LIN {X 0,Y 162.27,Z 688.109,A -85,B 0,C 180,E1 -25954.265,E2 -25954.265} C_VEL
LIN {X 0,Y 156.818,Z 700.099,A -85,B 0,C 180,E1 -25956.224,E2 -25956.224} C_VEL
LIN {X 0,Y 150.778,Z 711.775,A -85,B 0,C 180,E1 -25958.67,E2 -25958.67} C_VEL
LIN {X 0,Y 143.94,Z 723.54,A -85,B 0,C 180,E1 -25961.874,E2 -25961.874} C_VEL
LIN {X 0,Y 137.759,Z 733.192,A -85,B 0,C 180,E1 -25965.296,E2 -25965.296} C_VEL
LIN {X 0,Y 132.844,Z 740.567,A -85,B 0,C 180,E1 -25968.599,E2 -25968.599} C_VEL
LIN {X 0,Y 126.818,Z 749.022,A -85,B 0,C 180,E1 -25973.433,E2 -25973.433} C_VEL
LIN {X 0,Y 121.728,Z 756.009,A -85,B 0,C 180,E1 -25978.692,E2 -25978.692} C_VEL
LIN {X 0,Y 117.214,Z 762.465,A -85,B 0,C 180,E1 -25985.182,E2 -25985.182} C_VEL
LIN {X 0,Y 114.114,Z 767.443,A -85,B 0,C 180,E1 -25992.063,E2 -25992.063} C_VEL
LIN {X 0,Y 112.508,Z 771.077,A -85,B 0,C 180,E1 -25999.197,E2 -25999.197} C_VEL
LIN {X 0,Y 112.216,Z 772.187,A -85,B 0,C 180,E1 -26002.183,E2 -26002.183} C_VEL
LIN {X 0,Y 111.418,Z 773.145,A -85,B 0,C 180,E1 -26005.137,E2 -26005.137} C_VEL
LIN {X 0,Y 109.742,Z 773.826,A -85,B 0,C 180,E1 -26008.075,E2 -26008.075} C_VEL
LIN {X 0,Y 106.019,Z 774.46,A -85,B 0,C 180,E1 -26014.176,E2 -26014.176} C_VEL
LIN {X 0,Y 105.123,Z 774.478,A -85,B 0,C 180,E1 -26017.421,E2 -26017.421} C_VEL
LIN {X 0,Y 105.117,Z 774.446,A -85,B 0,C 180,E1 -26018.519,E2 -26018.519} C_VEL
LIN {X 0,Y 106.239,Z 773.913,A -85,B 0,C 180,E1 -26025.342,E2 -26025.342} C_VEL
LIN {X 0,Y 108.989,Z 772.261,A -85,B 0,C 180,E1 -26032.759,E2 -26032.759} C_VEL
LIN {X 0,Y 113.268,Z 769.502,A -85,B 0,C 180,E1 -26039.758,E2 -26039.758} C_VEL
LIN {X 0,Y 119.195,Z 765.541,A -85,B 0,C 180,E1 -26046.127,E2 -26046.127} C_VEL
LIN {X 0,Y 126.402,Z 760.299,A -85,B 0,C 180,E1 -26051.849,E2 -26051.849} C_VEL
LIN {X 0,Y 132.654,Z 755.491,A -85,B 0,C 180,E1 -26055.659,E2 -26055.659} C_VEL
LIN {X 0,Y 139.26,Z 749.833,A -85,B 0,C 180,E1 -26059.197,E2 -26059.197} C_VEL
LIN {X 0,Y 147.754,Z 742.03,A -85,B 0,C 180,E1 -26062.815,E2 -26062.815} C_VEL
LIN {X 0,Y 156.831,Z 732.723,A -85,B 0,C 180,E1 -26065.996,E2 -26065.996} C_VEL
LIN {X 0,Y 166.319,Z 721.594,A -85,B 0,C 180,E1 -26068.832,E2 -26068.832} C_VEL
LIN {X 0,Y 174.952,Z 709.953,A -85,B 0,C 180,E1 -26071.034,E2 -26071.034} C_VEL
LIN {X 0,Y 182.722,Z 697.753,A -85,B 0,C 180,E1 -26072.801,E2 -26072.801} C_VEL
LIN {X 0,Y 190.165,Z 683.997,A -85,B 0,C 180,E1 -26074.264,E2 -26074.264} C_VEL
LIN {X 0,Y 196.216,Z 670.493,A -85,B 0,C 180,E1 -26075.346,E2 -26075.346} C_VEL
LIN {X 0,Y 201.613,Z 655.52,A -85,B 0,C 180,E1 -26076.208,E2 -26076.208} C_VEL
LIN {X 0,Y 205.675,Z 640.602,A -85,B 0,C 180,E1 -26076.834,E2 -26076.834} C_VEL
LIN {X 0,Y 208.57,Z 625.043,A -85,B 0,C 180,E1 -26077.319,E2 -26077.319} C_VEL
LIN {X 0,Y 212.506,Z 591.895,A -85,B 0,C 180,E1 -26078.08,E2 -26078.08} C_VEL
LIN {X 0,Y 212.507,Z 590.897,A -85,B 0,C 180,E1 -26078.239,E2 -26078.239} C_VEL
LIN {X 0,Y 211.324,Z 586.522,A -85,B 0,C 180,E1 -26080.576,E2 -26080.576} C_VEL
LIN {X 0,Y 210.411,Z 584.182,A -85,B 0,C 180,E1 -26082.713,E2 -26082.713} C_VEL
LIN {X 0,Y 209.577,Z 581.413,A -85,B 0,C 180,E1 -26085.936,E2 -26085.936} C_VEL
LIN {X 0,Y 209.392,Z 581.09,A -85,B 0,C 180,E1 -26091.357,E2 -26091.357} C_VEL
LIN {X 0,Y 209.849,Z 581.667,A -85,B 0,C 180,E1 -26093.618,E2 -26093.618} C_VEL
LIN {X 0,Y 210.87,Z 584.782,A -85,B 0,C 180,E1 -26096.775,E2 -26096.775} C_VEL
LIN {X 0,Y 212.084,Z 588.141,A -85,B 0,C 180,E1 -26099.239,E2 -26099.239} C_VEL
LIN {X 0,Y 212.657,Z 589.826,A -85,B 0,C 180,E1 -26100.228,E2 -26100.228} C_VEL
LIN {X 0,Y 208.507,Z 624.685,A -85,B 0,C 180,E1 -26101.085,E2 -26101.085} C_VEL
LIN {X 0,Y 205.294,Z 640.714,A -85,B 0,C 180,E1 -26101.638,E2 -26101.638} C_VEL
LIN {X 0,Y 201.171,Z 655.223,A -85,B 0,C 180,E1 -26102.378,E2 -26102.378} C_VEL
LIN {X 0,Y 196.293,Z 668.552,A -85,B 0,C 180,E1 -26103.305,E2 -26103.305} C_VEL
LIN {X 0,Y 190.338,Z 681.794,A -85,B 0,C 180,E1 -26104.505,E2 -26104.505} C_VEL
LIN {X 0,Y 183.705,Z 694.085,A -85,B 0,C 180,E1 -26105.93,E2 -26105.93} C_VEL
LIN {X 0,Y 175.584,Z 706.828,A -85,B 0,C 180,E1 -26107.855,E2 -26107.855} C_VEL
LIN {X 0,Y 167.216,Z 718.068,A -85,B 0,C 180,E1 -26110.098,E2 -26110.098} C_VEL
LIN {X 0,Y 158.433,Z 728.344,A -85,B 0,C 180,E1 -26112.815,E2 -26112.815} C_VEL
LIN {X 0,Y 150.176,Z 736.866,A -85,B 0,C 180,E1 -26115.766,E2 -26115.766} C_VEL
LIN {X 0,Y 141.593,Z 744.777,A -85,B 0,C 180,E1 -26119.433,E2 -26119.433} C_VEL
LIN {X 0,Y 133.986,Z 751.07,A -85,B 0,C 180,E1 -26123.38,E2 -26123.38} C_VEL
LIN {X 0,Y 127.018,Z 756.227,A -85,B 0,C 180,E1 -26127.717,E2 -26127.717} C_VEL
LIN {X 0,Y 119.049,Z 761.614,A -85,B 0,C 180,E1 -26134.266,E2 -26134.266} C_VEL
LIN {X 0,Y 112.744,Z 765.391,A -85,B 0,C 180,E1 -26141.584,E2 -26141.584} C_VEL
LIN {X 0,Y 108.265,Z 767.673,A -85,B 0,C 180,E1 -26149.526,E2 -26149.526} C_VEL
LIN {X 0,Y 106.746,Z 768.28,A -85,B 0,C 180,E1 -26153.665,E2 -26153.665} C_VEL
LIN {X 0,Y 104.873,Z 768.47,A -85,B 0,C 180,E1 -26162.027,E2 -26162.027} C_VEL
LIN {X 0,Y 104.581,Z 767.341,A -85,B 0,C 180,E1 -26170.369,E2 -26170.369} C_VEL
LIN {X 0,Y 105.511,Z 764.943,A -85,B 0,C 180,E1 -26178.475,E2 -26178.475} C_VEL
LIN {X 0,Y 107.833,Z 761.254,A -85,B 0,C 180,E1 -26186.265,E2 -26186.265} C_VEL
LIN {X 0,Y 111.497,Z 756.221,A -85,B 0,C 180,E1 -26193.616,E2 -26193.616} C_VEL
LIN {X 0,Y 116.552,Z 749.716,A -85,B 0,C 180,E1 -26200.424,E2 -26200.424} C_VEL
LIN {X 0,Y 122.88,Z 741.548,A -85,B 0,C 180,E1 -26206.619,E2 -26206.619} C_VEL
LIN {X 0,Y 129.598,Z 732.606,A -85,B 0,C 180,E1 -26211.591,E2 -26211.591} C_VEL
LIN {X 0,Y 136.703,Z 722.284,A -85,B 0,C 180,E1 -26215.913,E2 -26215.913} C_VEL
LIN {X 0,Y 143.55,Z 711.455,A -85,B 0,C 180,E1 -26219.315,E2 -26219.315} C_VEL
LIN {X 0,Y 149.892,Z 700.19,A -85,B 0,C 180,E1 -26222.052,E2 -26222.052} C_VEL
LIN {X 0,Y 155.789,Z 688.229,A -85,B 0,C 180,E1 -26224.327,E2 -26224.327} C_VEL
LIN {X 0,Y 161.578,Z 674.427,A -85,B 0,C 180,E1 -26226.345,E2 -26226.345} C_VEL
LIN {X 0,Y 166.501,Z 660.122,A -85,B 0,C 180,E1 -26227.93,E2 -26227.93} C_VEL
LIN {X 0,Y 170.494,Z 645.425,A -85,B 0,C 180,E1 -26229.14,E2 -26229.14} C_VEL
LIN {X 0,Y 173.566,Z 630.355,A -85,B 0,C 180,E1 -26230.003,E2 -26230.003} C_VEL
LIN {X 0,Y 175.616,Z 614.874,A -85,B 0,C 180,E1 -26230.579,E2 -26230.579} C_VEL
LIN {X 0,Y 179.888,Z 570.202,A -85,B 0,C 180,E1 -26231.913,E2 -26231.913} C_VEL
LIN {X 0,Y 175.254,Z 560.703,A -85,B 0,C 180,E1 -26235.116,E2 -26235.116} C_VEL
LIN {X 0,Y 170.607,Z 551.973,A -85,B 0,C 180,E1 -26238.768,E2 -26238.768} C_VEL
LIN {X 0,Y 166.633,Z 545.183,A -85,B 0,C 180,E1 -26242.353,E2 -26242.353} C_VEL
LIN {X 0,Y 162.91,Z 538.962,A -85,B 0,C 180,E1 -26246.341,E2 -26246.341} C_VEL
LIN {X 0,Y 160.106,Z 534.703,A -85,B 0,C 180,E1 -26249.973,E2 -26249.973} C_VEL
LIN {X 0,Y 157.882,Z 531.017,A -85,B 0,C 180,E1 -26253.567,E2 -26253.567} C_VEL
LIN {X 0,Y 155.656,Z 528.166,A -85,B 0,C 180,E1 -26258.239,E2 -26258.239} C_VEL
LIN {X 0,Y 154.958,Z 526.341,A -85,B 0,C 180,E1 -26260.612,E2 -26260.612} C_VEL
LIN {X 0,Y 153.708,Z 525.25,A -85,B 0,C 180,E1 -26269.461,E2 -26269.461} C_VEL
LIN {X 0,Y 155.276,Z 526.167,A -85,B 0,C 180,E1 -26277.794,E2 -26277.794} C_VEL
LIN {X 0,Y 156.881,Z 529.591,A -85,B 0,C 180,E1 -26282.071,E2 -26282.071} C_VEL
LIN {X 0,Y 158.186,Z 531.195,A -85,B 0,C 180,E1 -26284.502,E2 -26284.502} C_VEL
LIN {X 0,Y 161.245,Z 536.157,A -85,B 0,C 180,E1 -26289.133,E2 -26289.133} C_VEL
LIN {X 0,Y 163.646,Z 540.079,A -85,B 0,C 180,E1 -26292.076,E2 -26292.076} C_VEL
LIN {X 0,Y 167.614,Z 546.604,A -85,B 0,C 180,E1 -26296.147,E2 -26296.147} C_VEL
LIN {X 0,Y 172.723,Z 555.773,A -85,B 0,C 180,E1 -26300.525,E2 -26300.525} C_VEL
LIN {X 0,Y 176.682,Z 565.689,A -85,B 0,C 180,E1 -26303.667,E2 -26303.667} C_VEL
LIN {X 0,Y 179.683,Z 573.874,A -85,B 0,C 180,E1 -26305.855,E2 -26305.855} C_VEL
LIN {X 0,Y 174.358,Z 628.461,A -85,B 0,C 180,E1 -26307.528,E2 -26307.528} C_VEL
LIN {X 0,Y 171.599,Z 644.728,A -85,B 0,C 180,E1 -26308.289,E2 -26308.289} C_VEL
LIN {X 0,Y 167.711,Z 660.014,A -85,B 0,C 180,E1 -26309.288,E2 -26309.288} C_VEL
LIN {X 0,Y 163.259,Z 673.839,A -85,B 0,C 180,E1 -26310.574,E2 -26310.574} C_VEL
LIN {X 0,Y 157.567,Z 688.206,A -85,B 0,C 180,E1 -26312.359,E2 -26312.359} C_VEL
LIN {X 0,Y 152.04,Z 699.961,A -85,B 0,C 180,E1 -26314.281,E2 -26314.281} C_VEL
LIN {X 0,Y 145.782,Z 711.627,A -85,B 0,C 180,E1 -26316.727,E2 -26316.727} C_VEL
LIN {X 0,Y 139.264,Z 722.481,A -85,B 0,C 180,E1 -26319.681,E2 -26319.681} C_VEL
LIN {X 0,Y 132.115,Z 733.155,A -85,B 0,C 180,E1 -26323.472,E2 -26323.472} C_VEL
LIN {X 0,Y 126.557,Z 741.051,A -85,B 0,C 180,E1 -26327.133,E2 -26327.133} C_VEL
LIN {X 0,Y 120.258,Z 749.409,A -85,B 0,C 180,E1 -26332.146,E2 -26332.146} C_VEL
LIN {X 0,Y 114.254,Z 757.19,A -85,B 0,C 180,E1 -26338.474,E2 -26338.474} C_VEL
LIN {X 0,Y 109.728,Z 763.354,A -85,B 0,C 180,E1 -26345.396,E2 -26345.396} C_VEL
LIN {X 0,Y 106.707,Z 768.064,A -85,B 0,C 180,E1 -26352.758,E2 -26352.758} C_VEL
LIN {X 0,Y 105.506,Z 770.697,A -85,B 0,C 180,E1 -26358.471,E2 -26358.471} C_VEL
LIN {X 0,Y 105.025,Z 773.144,A -85,B 0,C 180,E1 -26366.161,E2 -26366.161} C_VEL
LIN {X 0,Y 105.17,Z 773.911,A -85,B 0,C 180,E1 -26369.998,E2 -26369.998} C_VEL
LIN {X 0,Y 105.065,Z 774.477,A -85,B 0,C 180,E1 -26377.686,E2 -26377.686} C_VEL
LIN {X 0,Y 105.117,Z 774.446,A -85,B 0,C 180,E1 -26378.519,E2 -26378.519} C_VEL
LIN {X 0,Y 104.822,Z 774.318,A -85,B 0,C 180,E1 -26381.736,E2 -26381.736} C_VEL
LIN {X 0,Y 103.146,Z 773.669,A -85,B 0,C 180,E1 -26387.113,E2 -26387.113} C_VEL
LIN {X 0,Y 102.255,Z 772.859,A -85,B 0,C 180,E1 -26391.511,E2 -26391.511} C_VEL
LIN {X 0,Y 102.734,Z 772.048,A -85,B 0,C 180,E1 -26394.785,E2 -26394.785} C_VEL
LIN {X 0,Y 103.222,Z 771.714,A -85,B 0,C 180,E1 -26395.837,E2 -26395.837} C_VEL
LIN {X 0,Y 107.112,Z 769.508,A -85,B 0,C 180,E1 -26401.659,E2 -26401.659} C_VEL
LIN {X 0,Y 113.484,Z 765.616,A -85,B 0,C 180,E1 -26408.262,E2 -26408.262} C_VEL
LIN {X 0,Y 121.191,Z 760.483,A -85,B 0,C 180,E1 -26414.095,E2 -26414.095} C_VEL
LIN {X 0,Y 127.761,Z 755.783,A -85,B 0,C 180,E1 -26417.952,E2 -26417.952} C_VEL
LIN {X 0,Y 135.963,Z 749.177,A -85,B 0,C 180,E1 -26422.022,E2 -26422.022} C_VEL
LIN {X 0,Y 144.893,Z 741.301,A -85,B 0,C 180,E1 -26425.542,E2 -26425.542} C_VEL
LIN {X 0,Y 154.379,Z 731.92,A -85,B 0,C 180,E1 -26428.6,E2 -26428.6} C_VEL
LIN {X 0,Y 162.791,Z 722.439,A -85,B 0,C 180,E1 -26430.95,E2 -26430.95} C_VEL
LIN {X 0,Y 171.714,Z 710.933,A -85,B 0,C 180,E1 -26433.094,E2 -26433.094} C_VEL
LIN {X 0,Y 179.638,Z 699.057,A -85,B 0,C 180,E1 -26434.781,E2 -26434.781} C_VEL
LIN {X 0,Y 187.239,Z 685.685,A -85,B 0,C 180,E1 -26436.189,E2 -26436.189} C_VEL
LIN {X 0,Y 193.416,Z 672.678,A -85,B 0,C 180,E1 -26437.22,E2 -26437.22} C_VEL
LIN {X 0,Y 199.307,Z 657.258,A -85,B 0,C 180,E1 -26438.095,E2 -26438.095} C_VEL
LIN {X 0,Y 203.637,Z 642.297,A -85,B 0,C 180,E1 -26438.718,E2 -26438.718} C_VEL
LIN {X 0,Y 206.792,Z 626.525,A -85,B 0,C 180,E1 -26439.195,E2 -26439.195} C_VEL
LIN {X 0,Y 210.593,Z 595.394,A -85,B 0,C 180,E1 -26439.918,E2 -26439.918} C_VEL
LIN {X 0,Y 209.902,Z 592.781,A -85,B 0,C 180,E1 -26441.508,E2 -26441.508} C_VEL
LIN {X 0,Y 209.298,Z 591.026,A -85,B 0,C 180,E1 -26443.144,E2 -26443.144} C_VEL
LIN {X 0,Y 208.568,Z 588.359,A -85,B 0,C 180,E1 -26446.357,E2 -26446.357} C_VEL
LIN {X 0,Y 208.457,Z 588.126,A -85,B 0,C 180,E1 -26451.318,E2 -26451.318} C_VEL
LIN {X 0,Y 208.824,Z 588.647,A -85,B 0,C 180,E1 -26453.301,E2 -26453.301} C_VEL
LIN {X 0,Y 209.657,Z 591.398,A -85,B 0,C 180,E1 -26456.156,E2 -26456.156} C_VEL
LIN {X 0,Y 210.654,Z 594.475,A -85,B 0,C 180,E1 -26458.462,E2 -26458.462} C_VEL
LIN {X 0,Y 206.791,Z 625.689,A -85,B 0,C 180,E1 -26459.203,E2 -26459.203} C_VEL
LIN {X 0,Y 203.613,Z 641.04,A -85,B 0,C 180,E1 -26459.71,E2 -26459.71} C_VEL
LIN {X 0,Y 199.438,Z 655.419,A -85,B 0,C 180,E1 -26460.411,E2 -26460.411} C_VEL
LIN {X 0,Y 194.192,Z 669.329,A -85,B 0,C 180,E1 -26461.332,E2 -26461.332} C_VEL
LIN {X 0,Y 187.31,Z 683.964,A -85,B 0,C 180,E1 -26462.621,E2 -26462.621} C_VEL
LIN {X 0,Y 180.102,Z 696.586,A -85,B 0,C 180,E1 -26464.089,E2 -26464.089} C_VEL
LIN {X 0,Y 172.2,Z 708.333,A -85,B 0,C 180,E1 -26465.855,E2 -26465.855} C_VEL
LIN {X 0,Y 163.275,Z 719.746,A -85,B 0,C 180,E1 -26468.119,E2 -26468.119} C_VEL
LIN {X 0,Y 153.473,Z 730.558,A -85,B 0,C 180,E1 -26471.017,E2 -26471.017} C_VEL
LIN {X 0,Y 144.718,Z 738.936,A -85,B 0,C 180,E1 -26474.054,E2 -26474.054} C_VEL
LIN {X 0,Y 134.897,Z 747.278,A -85,B 0,C 180,E1 -26478.216,E2 -26478.216} C_VEL
LIN {X 0,Y 125.712,Z 754.118,A -85,B 0,C 180,E1 -26483.039,E2 -26483.039} C_VEL
LIN {X 0,Y 117.547,Z 759.504,A -85,B 0,C 180,E1 -26488.576,E2 -26488.576} C_VEL
LIN {X 0,Y 110.557,Z 763.601,A -85,B 0,C 180,E1 -26494.899,E2 -26494.899} C_VEL
LIN {X 0,Y 104.674,Z 766.617,A -85,B 0,C 180,E1 -26502.395,E2 -26502.395} C_VEL
LIN {X 0,Y 100.448,Z 768.371,A -85,B 0,C 180,E1 -26510.976,E2 -26510.976} C_VEL
LIN {X 0,Y 98.076,Z 768.74,A -85,B 0,C 180,E1 -26519.896,E2 -26519.896} C_VEL
LIN {X 0,Y 97.402,Z 767.787,A -85,B 0,C 180,E1 -26528.855,E2 -26528.855} C_VEL
LIN {X 0,Y 98.214,Z 765.558,A -85,B 0,C 180,E1 -26537.606,E2 -26537.606} C_VEL
LIN {X 0,Y 100.489,Z 762.048,A -85,B 0,C 180,E1 -26545.992,E2 -26545.992} C_VEL
LIN {X 0,Y 104.215,Z 757.199,A -85,B 0,C 180,E1 -26553.869,E2 -26553.869} C_VEL
LIN {X 0,Y 109.425,Z 750.895,A -85,B 0,C 180,E1 -26561.111,E2 -26561.111} C_VEL
LIN {X 0,Y 115.926,Z 742.959,A -85,B 0,C 180,E1 -26567.647,E2 -26567.647} C_VEL
LIN {X 0,Y 123.042,Z 734.077,A -85,B 0,C 180,E1 -26572.919,E2 -26572.919} C_VEL
LIN {X 0,Y 130.224,Z 724.224,A -85,B 0,C 180,E1 -26577.307,E2 -26577.307} C_VEL
LIN {X 0,Y 137.266,Z 713.734,A -85,B 0,C 180,E1 -26580.798,E2 -26580.798} C_VEL
LIN {X 0,Y 144.347,Z 701.867,A -85,B 0,C 180,E1 -26583.791,E2 -26583.791} C_VEL
LIN {X 0,Y 151.211,Z 688.531,A -85,B 0,C 180,E1 -26586.343,E2 -26586.343} C_VEL
LIN {X 0,Y 157.19,Z 674.745,A -85,B 0,C 180,E1 -26588.343,E2 -26588.343} C_VEL
LIN {X 0,Y 162.259,Z 660.473,A -85,B 0,C 180,E1 -26589.911,E2 -26589.911} C_VEL
LIN {X 0,Y 166.382,Z 645.806,A -85,B 0,C 180,E1 -26591.1,E2 -26591.1} C_VEL
LIN {X 0,Y 169.651,Z 630.125,A -85,B 0,C 180,E1 -26591.976,E2 -26591.976} C_VEL
LIN {X 0,Y 171.783,Z 614.022,A -85,B 0,C 180,E1 -26592.562,E2 -26592.562} C_VEL
LIN {X 0,Y 175.811,Z 573.246,A -85,B 0,C 180,E1 -26593.758,E2 -26593.758} C_VEL
LIN {X 0,Y 171.013,Z 563.284,A -85,B 0,C 180,E1 -26597.435,E2 -26597.435} C_VEL
LIN {X 0,Y 166.752,Z 555.193,A -85,B 0,C 180,E1 -26601.149,E2 -26601.149} C_VEL
LIN {X 0,Y 162.967,Z 548.616,A -85,B 0,C 180,E1 -26605.024,E2 -26605.024} C_VEL
LIN {X 0,Y 160.575,Z 544.605,A -85,B 0,C 180,E1 -26607.91,E2 -26607.91} C_VEL
LIN {X 0,Y 158.639,Z 541.417,A -85,B 0,C 180,E1 -26610.622,E2 -26610.622} C_VEL
LIN {X 0,Y 156.447,Z 537.738,A -85,B 0,C 180,E1 -26614.394,E2 -26614.394} C_VEL
LIN {X 0,Y 154.399,Z 534.759,A -85,B 0,C 180,E1 -26619.116,E2 -26619.116} C_VEL
LIN {X 0,Y 153.931,Z 533.338,A -85,B 0,C 180,E1 -26620.919,E2 -26620.919} C_VEL
LIN {X 0,Y 152.781,Z 532.297,A -85,B 0,C 180,E1 -26629.396,E2 -26629.396} C_VEL
LIN {X 0,Y 154.192,Z 533.209,A -85,B 0,C 180,E1 -26637.387,E2 -26637.387} C_VEL
LIN {X 0,Y 155.821,Z 536.604,A -85,B 0,C 180,E1 -26641.85,E2 -26641.85} C_VEL
LIN {X 0,Y 156.819,Z 537.928,A -85,B 0,C 180,E1 -26643.819,E2 -26643.819} C_VEL
LIN {X 0,Y 159.645,Z 542.727,A -85,B 0,C 180,E1 -26648.351,E2 -26648.351} C_VEL
LIN {X 0,Y 161.934,Z 546.701,A -85,B 0,C 180,E1 -26651.342,E2 -26651.342} C_VEL
LIN {X 0,Y 165.674,Z 553.156,A -85,B 0,C 180,E1 -26655.374,E2 -26655.374} C_VEL
LIN {X 0,Y 170.163,Z 561.536,A -85,B 0,C 180,E1 -26659.44,E2 -26659.44} C_VEL
LIN {X 0,Y 174.602,Z 573.496,A -85,B 0,C 180,E1 -26663.185,E2 -26663.185} C_VEL
LIN {X 0,Y 175.69,Z 576.563,A -85,B 0,C 180,E1 -26664.028,E2 -26664.028} C_VEL
LIN {X 0,Y 170.252,Z 629.604,A -85,B 0,C 180,E1 -26665.615,E2 -26665.615} C_VEL
LIN {X 0,Y 167.411,Z 645.329,A -85,B 0,C 180,E1 -26666.358,E2 -26666.358} C_VEL
LIN {X 0,Y 163.599,Z 659.829,A -85,B 0,C 180,E1 -26667.287,E2 -26667.287} C_VEL
LIN {X 0,Y 159.018,Z 673.653,A -85,B 0,C 180,E1 -26668.549,E2 -26668.549} C_VEL
LIN {X 0,Y 153.073,Z 688.196,A -85,B 0,C 180,E1 -26670.333,E2 -26670.333} C_VEL
LIN {X 0,Y 147.448,Z 699.78,A -85,B 0,C 180,E1 -26672.215,E2 -26672.215} C_VEL
LIN {X 0,Y 140.967,Z 711.447,A -85,B 0,C 180,E1 -26674.65,E2 -26674.65} C_VEL
LIN {X 0,Y 133.574,Z 723.205,A -85,B 0,C 180,E1 -26677.885,E2 -26677.885} C_VEL
LIN {X 0,Y 126.415,Z 733.377,A -85,B 0,C 180,E1 -26681.602,E2 -26681.602} C_VEL
LIN {X 0,Y 120.359,Z 741.498,A -85,B 0,C 180,E1 -26685.515,E2 -26685.515} C_VEL
LIN {X 0,Y 114.677,Z 748.667,A -85,B 0,C 180,E1 -26689.945,E2 -26689.945} C_VEL
LIN {X 0,Y 108.199,Z 756.568,A -85,B 0,C 180,E1 -26696.486,E2 -26696.486} C_VEL
LIN {X 0,Y 103.243,Z 762.818,A -85,B 0,C 180,E1 -26703.736,E2 -26703.736} C_VEL
LIN {X 0,Y 99.894,Z 767.602,A -85,B 0,C 180,E1 -26711.541,E2 -26711.541} C_VEL
LIN {X 0,Y 98.502,Z 770.315,A -85,B 0,C 180,E1 -26717.638,E2 -26717.638} C_VEL
LIN {X 0,Y 97.927,Z 772.84,A -85,B 0,C 180,E1 -26725.882,E2 -26725.882} C_VEL
LIN {X 0,Y 98.073,Z 773.626,A -85,B 0,C 180,E1 -26729.998,E2 -26729.998} C_VEL
LIN {X 0,Y 98.016,Z 774.249,A -85,B 0,C 180,E1 -26738.243,E2 -26738.243} C_VEL
LIN {X 0,Y 99.341,Z 773.765,A -85,B 0,C 180,E1 -26746.436,E2 -26746.436} C_VEL
LIN {X 0,Y 102.406,Z 772.195,A -85,B 0,C 180,E1 -26754.313,E2 -26754.313} C_VEL
LIN {X 0,Y 103.222,Z 771.714,A -85,B 0,C 180,E1 -26755.837,E2 -26755.837} C_VEL
LIN {X 0,Y 104.467,Z 770.705,A -85,B 0,C 180,E1 -26758.974,E2 -26758.974} C_VEL
LIN {X 0,Y 105.464,Z 768.728,A -85,B 0,C 180,E1 -26764.257,E2 -26764.257} C_VEL
LIN {X 0,Y 107.291,Z 766.389,A -85,B 0,C 180,E1 -26769.355,E2 -26769.355} C_VEL
LIN {X 0,Y 109.734,Z 764.681,A -85,B 0,C 180,E1 -26772.054,E2 -26772.054} C_VEL
LIN {X 0,Y 118.478,Z 759.24,A -85,B 0,C 180,E1 -26777.855,E2 -26777.855} C_VEL
LIN {X 0,Y 128.989,Z 751.672,A -85,B 0,C 180,E1 -26783.331,E2 -26783.331} C_VEL
LIN {X 0,Y 139.649,Z 743.039,A -85,B 0,C 180,E1 -26787.45,E2 -26787.45} C_VEL
LIN {X 0,Y 149.402,Z 734.054,A -85,B 0,C 180,E1 -26790.484,E2 -26790.484} C_VEL
LIN {X 0,Y 159.494,Z 723.293,A -85,B 0,C 180,E1 -26793.159,E2 -26793.159} C_VEL
LIN {X 0,Y 168.754,Z 711.903,A -85,B 0,C 180,E1 -26795.242,E2 -26795.242} C_VEL
LIN {X 0,Y 177.541,Z 699.225,A -85,B 0,C 180,E1 -26796.974,E2 -26796.974} C_VEL
LIN {X 0,Y 185.318,Z 685.937,A -85,B 0,C 180,E1 -26798.296,E2 -26798.296} C_VEL
LIN {X 0,Y 191.623,Z 672.986,A -85,B 0,C 180,E1 -26799.262,E2 -26799.262} C_VEL
LIN {X 0,Y 197.622,Z 657.768,A -85,B 0,C 180,E1 -26800.079,E2 -26800.079} C_VEL
LIN {X 0,Y 202.284,Z 642.024,A -85,B 0,C 180,E1 -26800.689,E2 -26800.689} C_VEL
LIN {X 0,Y 205.452,Z 626.585,A -85,B 0,C 180,E1 -26801.128,E2 -26801.128} C_VEL
LIN {X 0,Y 208.827,Z 599.844,A -85,B 0,C 180,E1 -26801.748,E2 -26801.748} C_VEL
LIN {X 0,Y 208.205,Z 597.884,A -85,B 0,C 180,E1 -26803.557,E2 -26803.557} C_VEL
LIN {X 0,Y 207.577,Z 595.346,A -85,B 0,C 180,E1 -26806.712,E2 -26806.712} C_VEL
LIN {X 0,Y 207.523,Z 595.162,A -85,B 0,C 180,E1 -26811.278,E2 -26811.278} C_VEL
LIN {X 0,Y 207.809,Z 595.517,A -85,B 0,C 180,E1 -26812.904,E2 -26812.904} C_VEL
LIN {X 0,Y 208.581,Z 598.435,A -85,B 0,C 180,E1 -26815.879,E2 -26815.879} C_VEL
LIN {X 0,Y 208.859,Z 599.466,A -85,B 0,C 180,E1 -26816.677,E2 -26816.677} C_VEL
LIN {X 0,Y 205.583,Z 625.132,A -85,B 0,C 180,E1 -26817.242,E2 -26817.242} C_VEL
LIN {X 0,Y 202.291,Z 640.93,A -85,B 0,C 180,E1 -26817.736,E2 -26817.736} C_VEL
LIN {X 0,Y 198.326,Z 654.413,A -85,B 0,C 180,E1 -26818.341,E2 -26818.341} C_VEL
LIN {X 0,Y 192.842,Z 668.902,A -85,B 0,C 180,E1 -26819.231,E2 -26819.231} C_VEL
LIN {X 0,Y 186.509,Z 682.3,A -85,B 0,C 180,E1 -26820.325,E2 -26820.325} C_VEL
LIN {X 0,Y 179.28,Z 694.961,A -85,B 0,C 180,E1 -26821.659,E2 -26821.659} C_VEL
LIN {X 0,Y 170.723,Z 707.562,A -85,B 0,C 180,E1 -26823.399,E2 -26823.399} C_VEL
LIN {X 0,Y 162.346,Z 718.131,A -85,B 0,C 180,E1 -26825.353,E2 -26825.353} C_VEL
LIN {X 0,Y 152.619,Z 728.75,A -85,B 0,C 180,E1 -26827.941,E2 -26827.941} C_VEL
LIN {X 0,Y 143.127,Z 737.731,A -85,B 0,C 180,E1 -26830.879,E2 -26830.879} C_VEL
LIN {X 0,Y 132.692,Z 746.349,A -85,B 0,C 180,E1 -26834.857,E2 -26834.857} C_VEL
LIN {X 0,Y 123.295,Z 753.126,A -85,B 0,C 180,E1 -26839.315,E2 -26839.315} C_VEL
LIN {X 0,Y 115.369,Z 758.193,A -85,B 0,C 180,E1 -26843.975,E2 -26843.975} C_VEL
LIN {X 0,Y 106.542,Z 763.148,A -85,B 0,C 180,E1 -26850.964,E2 -26850.964} C_VEL
LIN {X 0,Y 99.451,Z 766.534,A -85,B 0,C 180,E1 -26858.986,E2 -26858.986} C_VEL
LIN {X 0,Y 94.253,Z 768.495,A -85,B 0,C 180,E1 -26868.217,E2 -26868.217} C_VEL
LIN {X 0,Y 91.263,Z 768.991,A -85,B 0,C 180,E1 -26877.899,E2 -26877.899} C_VEL
LIN {X 0,Y 90.282,Z 768.223,A -85,B 0,C 180,E1 -26887.097,E2 -26887.097} C_VEL
LIN {X 0,Y 90.412,Z 767.339,A -85,B 0,C 180,E1 -26891.887,E2 -26891.887} C_VEL
LIN {X 0,Y 91.799,Z 764.615,A -85,B 0,C 180,E1 -26901.195,E2 -26901.195} C_VEL
LIN {X 0,Y 94.8,Z 760.595,A -85,B 0,C 180,E1 -26910.002,E2 -26910.002} C_VEL
LIN {X 0,Y 99.393,Z 755.213,A -85,B 0,C 180,E1 -26918.132,E2 -26918.132} C_VEL
LIN {X 0,Y 105.505,Z 748.331,A -85,B 0,C 180,E1 -26925.455,E2 -26925.455} C_VEL
LIN {X 0,Y 111.925,Z 740.894,A -85,B 0,C 180,E1 -26931.167,E2 -26931.167} C_VEL
LIN {X 0,Y 119.335,Z 731.92,A -85,B 0,C 180,E1 -26936.214,E2 -26936.214} C_VEL
LIN {X 0,Y 126.23,Z 722.79,A -85,B 0,C 180,E1 -26940.073,E2 -26940.073} C_VEL
LIN {X 0,Y 133.681,Z 711.97,A -85,B 0,C 180,E1 -26943.507,E2 -26943.507} C_VEL
LIN {X 0,Y 140.521,Z 700.71,A -85,B 0,C 180,E1 -26946.238,E2 -26946.238} C_VEL
LIN {X 0,Y 146.84,Z 688.779,A -85,B 0,C 180,E1 -26948.478,E2 -26948.478} C_VEL
LIN {X 0,Y 152.999,Z 675.014,A -85,B 0,C 180,E1 -26950.455,E2 -26950.455} C_VEL
LIN {X 0,Y 158.237,Z 660.75,A -85,B 0,C 180,E1 -26951.991,E2 -26951.991} C_VEL
LIN {X 0,Y 162.645,Z 645.372,A -85,B 0,C 180,E1 -26953.207,E2 -26953.207} C_VEL
LIN {X 0,Y 165.872,Z 630.234,A -85,B 0,C 180,E1 -26954.025,E2 -26954.025} C_VEL
LIN {X 0,Y 168.017,Z 614.613,A -85,B 0,C 180,E1 -26954.58,E2 -26954.58} C_VEL
LIN {X 0,Y 171.889,Z 576.49,A -85,B 0,C 180,E1 -26955.685,E2 -26955.685} C_VEL
LIN {X 0,Y 167.301,Z 566.697,A -85,B 0,C 180,E1 -26959.543,E2 -26959.543} C_VEL
LIN {X 0,Y 163.227,Z 558.743,A -85,B 0,C 180,E1 -26963.557,E2 -26963.557} C_VEL
LIN {X 0,Y 159.282,Z 551.65,A -85,B 0,C 180,E1 -26968.254,E2 -26968.254} C_VEL
LIN {X 0,Y 157.15,Z 548.075,A -85,B 0,C 180,E1 -26971.348,E2 -26971.348} C_VEL
LIN {X 0,Y 155.103,Z 544.481,A -85,B 0,C 180,E1 -26975.13,E2 -26975.13} C_VEL
LIN {X 0,Y 153.206,Z 541.433,A -85,B 0,C 180,E1 -26979.902,E2 -26979.902} C_VEL
LIN {X 0,Y 152.906,Z 540.329,A -85,B 0,C 180,E1 -26981.231,E2 -26981.231} C_VEL
LIN {X 0,Y 151.855,Z 539.319,A -85,B 0,C 180,E1 -26989.331,E2 -26989.331} C_VEL
LIN {X 0,Y 153.1,Z 540.136,A -85,B 0,C 180,E1 -26996.889,E2 -26996.889} C_VEL
LIN {X 0,Y 154.667,Z 543.503,A -85,B 0,C 180,E1 -27001.439,E2 -27001.439} C_VEL
LIN {X 0,Y 155.496,Z 544.722,A -85,B 0,C 180,E1 -27003.176,E2 -27003.176} C_VEL
LIN {X 0,Y 158.131,Z 549.436,A -85,B 0,C 180,E1 -27007.662,E2 -27007.662} C_VEL
LIN {X 0,Y 160.165,Z 553.133,A -85,B 0,C 180,E1 -27010.479,E2 -27010.479} C_VEL
LIN {X 0,Y 163.714,Z 559.588,A -85,B 0,C 180,E1 -27014.528,E2 -27014.528} C_VEL
LIN {X 0,Y 167.472,Z 567.031,A -85,B 0,C 180,E1 -27018.186,E2 -27018.186} C_VEL
LIN {X 0,Y 171.143,Z 577.375,A -85,B 0,C 180,E1 -27021.531,E2 -27021.531} C_VEL
LIN {X 0,Y 171.796,Z 579.348,A -85,B 0,C 180,E1 -27022.095,E2 -27022.095} C_VEL
LIN {X 0,Y 166.461,Z 629.665,A -85,B 0,C 180,E1 -27023.582,E2 -27023.582} C_VEL
LIN {X 0,Y 163.585,Z 645.099,A -85,B 0,C 180,E1 -27024.291,E2 -27024.291} C_VEL
LIN {X 0,Y 159.347,Z 660.688,A -85,B 0,C 180,E1 -27025.289,E2 -27025.289} C_VEL
LIN {X 0,Y 154.287,Z 675.22,A -85,B 0,C 180,E1 -27026.624,E2 -27026.624} C_VEL
LIN {X 0,Y 148.345,Z 689.06,A -85,B 0,C 180,E1 -27028.34,E2 -27028.34} C_VEL
LIN {X 0,Y 142.341,Z 700.819,A -85,B 0,C 180,E1 -27030.223,E2 -27030.223} C_VEL
LIN {X 0,Y 135.018,Z 713.366,A -85,B 0,C 180,E1 -27032.927,E2 -27032.927} C_VEL
LIN {X 0,Y 128.021,Z 723.872,A -85,B 0,C 180,E1 -27035.928,E2 -27035.928} C_VEL
LIN {X 0,Y 120.829,Z 733.601,A -85,B 0,C 180,E1 -27039.582,E2 -27039.582} C_VEL
LIN {X 0,Y 113.277,Z 743.165,A -85,B 0,C 180,E1 -27044.478,E2 -27044.478} C_VEL
LIN {X 0,Y 106.479,Z 751.074,A -85,B 0,C 180,E1 -27049.942,E2 -27049.942} C_VEL
LIN {X 0,Y 100.762,Z 757.61,A -85,B 0,C 180,E1 -27056.081,E2 -27056.081} C_VEL
LIN {X 0,Y 95.747,Z 763.586,A -85,B 0,C 180,E1 -27063.868,E2 -27063.868} C_VEL
LIN {X 0,Y 92.466,Z 768.138,A -85,B 0,C 180,E1 -27072.298,E2 -27072.298} C_VEL
LIN {X 0,Y 91.025,Z 771.378,A -85,B 0,C 180,E1 -27081.115,E2 -27081.115} C_VEL
LIN {X 0,Y 90.97,Z 773.315,A -85,B 0,C 180,E1 -27089.998,E2 -27089.998} C_VEL
LIN {X 0,Y 90.962,Z 774.018,A -85,B 0,C 180,E1 -27098.887,E2 -27098.887} C_VEL
LIN {X 0,Y 92.488,Z 773.616,A -85,B 0,C 180,E1 -27107.692,E2 -27107.692} C_VEL
LIN {X 0,Y 96.474,Z 771.836,A -85,B 0,C 180,E1 -27117.104,E2 -27117.104} C_VEL
LIN {X 0,Y 101.091,Z 769.502,A -85,B 0,C 180,E1 -27123.788,E2 -27123.788} C_VEL
LIN {X 0,Y 107.959,Z 765.702,A -85,B 0,C 180,E1 -27130.613,E2 -27130.613} C_VEL
LIN {X 0,Y 109.734,Z 764.681,A -85,B 0,C 180,E1 -27132.054,E2 -27132.054} C_VEL
LIN {X 0,Y 112.397,Z 762.87,A -85,B 0,C 180,E1 -27134.618,E2 -27134.618} C_VEL
LIN {X 0,Y 115.715,Z 759.649,A -85,B 0,C 180,E1 -27139.04,E2 -27139.04} C_VEL
LIN {X 0,Y 119.547,Z 755.97,A -85,B 0,C 180,E1 -27143.128,E2 -27143.128} C_VEL
LIN {X 0,Y 122.876,Z 753.414,A -85,B 0,C 180,E1 -27145.103,E2 -27145.103} C_VEL
LIN {X 0,Y 133.161,Z 745.772,A -85,B 0,C 180,E1 -27149.049,E2 -27149.049} C_VEL
LIN {X 0,Y 143.104,Z 737.376,A -85,B 0,C 180,E1 -27152.124,E2 -27152.124} C_VEL
LIN {X 0,Y 153.413,Z 727.361,A -85,B 0,C 180,E1 -27154.787,E2 -27154.787} C_VEL
LIN {X 0,Y 163.49,Z 716.002,A -85,B 0,C 180,E1 -27156.95,E2 -27156.95} C_VEL
LIN {X 0,Y 171.819,Z 705.109,A -85,B 0,C 180,E1 -27158.515,E2 -27158.515} C_VEL
LIN {X 0,Y 179.689,Z 693.087,A -85,B 0,C 180,E1 -27159.827,E2 -27159.827} C_VEL
LIN {X 0,Y 186.848,Z 680.096,A -85,B 0,C 180,E1 -27160.91,E2 -27160.91} C_VEL
LIN {X 0,Y 193.333,Z 665.837,A -85,B 0,C 180,E1 -27161.743,E2 -27161.743} C_VEL
LIN {X 0,Y 198.623,Z 651.033,A -85,B 0,C 180,E1 -27162.386,E2 -27162.386} C_VEL
LIN {X 0,Y 202.711,Z 635.535,A -85,B 0,C 180,E1 -27162.877,E2 -27162.877} C_VEL
LIN {X 0,Y 205.504,Z 619.272,A -85,B 0,C 180,E1 -27163.243,E2 -27163.243} C_VEL
LIN {X 0,Y 207.256,Z 605.056,A -85,B 0,C 180,E1 -27163.553,E2 -27163.553} C_VEL
LIN {X 0,Y 206.594,Z 602.334,A -85,B 0,C 180,E1 -27167.07,E2 -27167.07} C_VEL
LIN {X 0,Y 206.526,Z 602.12,A -85,B 0,C 180,E1 -27170.69,E2 -27170.69} C_VEL
LIN {X 0,Y 206.821,Z 602.583,A -85,B 0,C 180,E1 -27172.686,E2 -27172.686} C_VEL
LIN {X 0,Y 207.291,Z 604.558,A -85,B 0,C 180,E1 -27174.844,E2 -27174.844} C_VEL
LIN {X 0,Y 204.496,Z 625.699,A -85,B 0,C 180,E1 -27175.291,E2 -27175.291} C_VEL
LIN {X 0,Y 201.08,Z 641.592,A -85,B 0,C 180,E1 -27175.76,E2 -27175.76} C_VEL
LIN {X 0,Y 196.721,Z 655.947,A -85,B 0,C 180,E1 -27176.377,E2 -27176.377} C_VEL
LIN {X 0,Y 190.849,Z 670.721,A -85,B 0,C 180,E1 -27177.246,E2 -27177.246} C_VEL
LIN {X 0,Y 183.951,Z 684.585,A -85,B 0,C 180,E1 -27178.345,E2 -27178.345} C_VEL
LIN {X 0,Y 175.695,Z 698.197,A -85,B 0,C 180,E1 -27179.774,E2 -27179.774} C_VEL
LIN {X 0,Y 166.961,Z 710.292,A -85,B 0,C 180,E1 -27181.449,E2 -27181.449} C_VEL
LIN {X 0,Y 158.391,Z 720.475,A -85,B 0,C 180,E1 -27183.325,E2 -27183.325} C_VEL
LIN {X 0,Y 148.356,Z 730.773,A -85,B 0,C 180,E1 -27185.852,E2 -27185.852} C_VEL
LIN {X 0,Y 138.496,Z 739.486,A -85,B 0,C 180,E1 -27188.757,E2 -27188.757} C_VEL
LIN {X 0,Y 127.642,Z 747.858,A -85,B 0,C 180,E1 -27192.724,E2 -27192.724} C_VEL
LIN {X 0,Y 117.432,Z 754.65,A -85,B 0,C 180,E1 -27197.413,E2 -27197.413} C_VEL
LIN {X 0,Y 107.283,Z 760.454,A -85,B 0,C 180,E1 -27203.498,E2 -27203.498} C_VEL
LIN {X 0,Y 98.358,Z 764.8,A -85,B 0,C 180,E1 -27210.975,E2 -27210.975} C_VEL
LIN {X 0,Y 91.317,Z 767.636,A -85,B 0,C 180,E1 -27219.684,E2 -27219.684} C_VEL
LIN {X 0,Y 86.447,Z 769.035,A -85,B 0,C 180,E1 -27229.433,E2 -27229.433} C_VEL
LIN {X 0,Y 83.774,Z 769.063,A -85,B 0,C 180,E1 -27239.781,E2 -27239.781} C_VEL
LIN {X 0,Y 83.244,Z 767.775,A -85,B 0,C 180,E1 -27250.266,E2 -27250.266} C_VEL
LIN {X 0,Y 84.433,Z 765.221,A -85,B 0,C 180,E1 -27260.42,E2 -27260.42} C_VEL
LIN {X 0,Y 87.461,Z 761.372,A -85,B 0,C 180,E1 -27270.003,E2 -27270.003} C_VEL
LIN {X 0,Y 92.186,Z 756.172,A -85,B 0,C 180,E1 -27278.773,E2 -27278.773} C_VEL
LIN {X 0,Y 98.526,Z 749.487,A -85,B 0,C 180,E1 -27286.58,E2 -27286.58} C_VEL
LIN {X 0,Y 105.229,Z 742.262,A -85,B 0,C 180,E1 -27292.585,E2 -27292.585} C_VEL
LIN {X 0,Y 112.894,Z 733.536,A -85,B 0,C 180,E1 -27297.835,E2 -27297.835} C_VEL
LIN {X 0,Y 121.273,Z 723.025,A -85,B 0,C 180,E1 -27302.417,E2 -27302.417} C_VEL
LIN {X 0,Y 129.042,Z 712.206,A -85,B 0,C 180,E1 -27305.838,E2 -27305.838} C_VEL
LIN {X 0,Y 136.426,Z 700.425,A -85,B 0,C 180,E1 -27308.656,E2 -27308.656} C_VEL
LIN {X 0,Y 143.379,Z 687.578,A -85,B 0,C 180,E1 -27310.967,E2 -27310.967} C_VEL
LIN {X 0,Y 149.735,Z 673.49,A -85,B 0,C 180,E1 -27312.89,E2 -27312.89} C_VEL
LIN {X 0,Y 155.152,Z 658.741,A -85,B 0,C 180,E1 -27314.371,E2 -27314.371} C_VEL
LIN {X 0,Y 159.485,Z 643.465,A -85,B 0,C 180,E1 -27315.494,E2 -27315.494} C_VEL
LIN {X 0,Y 162.737,Z 627.624,A -85,B 0,C 180,E1 -27316.282,E2 -27316.282} C_VEL
LIN {X 0,Y 165.093,Z 608.944,A -85,B 0,C 180,E1 -27316.872,E2 -27316.872} C_VEL
LIN {X 0,Y 168.187,Z 579.867,A -85,B 0,C 180,E1 -27317.661,E2 -27317.661} C_VEL
LIN {X 0,Y 164.342,Z 571.419,A -85,B 0,C 180,E1 -27321.2,E2 -27321.2} C_VEL
LIN {X 0,Y 161.031,Z 564.638,A -85,B 0,C 180,E1 -27324.73,E2 -27324.73} C_VEL
LIN {X 0,Y 157.484,Z 557.889,A -85,B 0,C 180,E1 -27329.31,E2 -27329.31} C_VEL
LIN {X 0,Y 155.473,Z 554.405,A -85,B 0,C 180,E1 -27332.45,E2 -27332.45} C_VEL
LIN {X 0,Y 153.845,Z 551.309,A -85,B 0,C 180,E1 -27335.723,E2 -27335.723} C_VEL
LIN {X 0,Y 152.047,Z 548.129,A -85,B 0,C 180,E1 -27340.674,E2 -27340.674} C_VEL
LIN {X 0,Y 151.801,Z 547.249,A -85,B 0,C 180,E1 -27341.883,E2 -27341.883} C_VEL
LIN {X 0,Y 150.925,Z 546.368,A -85,B 0,C 180,E1 -27349.264,E2 -27349.264} C_VEL
LIN {X 0,Y 152.015,Z 547.101,A -85,B 0,C 180,E1 -27356.384,E2 -27356.384} C_VEL
LIN {X 0,Y 153.707,Z 550.676,A -85,B 0,C 180,E1 -27361.448,E2 -27361.448} C_VEL
LIN {X 0,Y 154.361,Z 551.923,A -85,B 0,C 180,E1 -27362.904,E2 -27362.904} C_VEL
LIN {X 0,Y 156.667,Z 556.189,A -85,B 0,C 180,E1 -27367.019,E2 -27367.019} C_VEL
LIN {X 0,Y 159.483,Z 561.524,A -85,B 0,C 180,E1 -27370.972,E2 -27370.972} C_VEL
LIN {X 0,Y 163.002,Z 568.51,A -85,B 0,C 180,E1 -27374.992,E2 -27374.992} C_VEL
LIN {X 0,Y 165.354,Z 573.8,A -85,B 0,C 180,E1 -27377.388,E2 -27377.388} C_VEL
LIN {X 0,Y 168.076,Z 582.056,A -85,B 0,C 180,E1 -27380.054,E2 -27380.054} C_VEL
LIN {X 0,Y 162.949,Z 629.367,A -85,B 0,C 180,E1 -27381.444,E2 -27381.444} C_VEL
LIN {X 0,Y 159.916,Z 645.165,A -85,B 0,C 180,E1 -27382.148,E2 -27382.148} C_VEL
LIN {X 0,Y 155.662,Z 660.401,A -85,B 0,C 180,E1 -27383.085,E2 -27383.085} C_VEL
LIN {X 0,Y 150.463,Z 674.952,A -85,B 0,C 180,E1 -27384.378,E2 -27384.378} C_VEL
LIN {X 0,Y 144.355,Z 688.776,A -85,B 0,C 180,E1 -27386.04,E2 -27386.04} C_VEL
LIN {X 0,Y 138.156,Z 700.57,A -85,B 0,C 180,E1 -27387.886,E2 -27387.886} C_VEL
LIN {X 0,Y 130.556,Z 713.12,A -85,B 0,C 180,E1 -27390.535,E2 -27390.535} C_VEL
LIN {X 0,Y 122.646,Z 724.542,A -85,B 0,C 180,E1 -27393.807,E2 -27393.807} C_VEL
LIN {X 0,Y 114.47,Z 734.996,A -85,B 0,C 180,E1 -27397.875,E2 -27397.875} C_VEL
LIN {X 0,Y 106.206,Z 744.806,A -85,B 0,C 180,E1 -27403.287,E2 -27403.287} C_VEL
LIN {X 0,Y 100.127,Z 751.366,A -85,B 0,C 180,E1 -27408.176,E2 -27408.176} C_VEL
LIN {X 0,Y 93.216,Z 758.745,A -85,B 0,C 180,E1 -27415.756,E2 -27415.756} C_VEL
LIN {X 0,Y 88.284,Z 764.321,A -85,B 0,C 180,E1 -27424.032,E2 -27424.032} C_VEL
LIN {X 0,Y 85.669,Z 767.696,A -85,B 0,C 180,E1 -27430.841,E2 -27430.841} C_VEL
LIN {X 0,Y 83.983,Z 770.991,A -85,B 0,C 180,E1 -27440.363,E2 -27440.363} C_VEL
LIN {X 0,Y 83.875,Z 773.005,A -85,B 0,C 180,E1 -27449.997,E2 -27449.997} C_VEL
LIN {X 0,Y 83.934,Z 773.789,A -85,B 0,C 180,E1 -27459.638,E2 -27459.638} C_VEL
LIN {X 0,Y 85.69,Z 773.472,A -85,B 0,C 180,E1 -27469.148,E2 -27469.148} C_VEL
LIN {X 0,Y 89.521,Z 772.063,A -85,B 0,C 180,E1 -27478.099,E2 -27478.099} C_VEL
LIN {X 0,Y 95.239,Z 769.494,A -85,B 0,C 180,E1 -27486.178,E2 -27486.178} C_VEL
LIN {X 0,Y 104.697,Z 764.724,A -85,B 0,C 180,E1 -27494.812,E2 -27494.812} C_VEL
LIN {X 0,Y 113.823,Z 759.46,A -85,B 0,C 180,E1 -27500.513,E2 -27500.513} C_VEL
LIN {X 0,Y 122.876,Z 753.414,A -85,B 0,C 180,E1 -27505.103,E2 -27505.103} C_VEL
LIN {X 0,Y 126.329,Z 750.769,A -85,B 0,C 180,E1 -27506.945,E2 -27506.945} C_VEL
LIN {X 0,Y 134.986,Z 742.499,A -85,B 0,C 180,E1 -27512.76,E2 -27512.76} C_VEL
LIN {X 0,Y 138.461,Z 739.325,A -85,B 0,C 180,E1 -27514.25,E2 -27514.25} C_VEL
LIN {X 0,Y 139.766,Z 738.186,A -85,B 0,C 180,E1 -27514.639,E2 -27514.639} C_VEL
LIN {X 0,Y 150.55,Z 728.195,A -85,B 0,C 180,E1 -27517.21,E2 -27517.21} C_VEL
LIN {X 0,Y 160.915,Z 717.008,A -85,B 0,C 180,E1 -27519.259,E2 -27519.259} C_VEL
LIN {X 0,Y 170.173,Z 705.324,A -85,B 0,C 180,E1 -27520.853,E2 -27520.853} C_VEL
LIN {X 0,Y 178.218,Z 693.382,A -85,B 0,C 180,E1 -27522.051,E2 -27522.051} C_VEL
LIN {X 0,Y 185.505,Z 680.502,A -85,B 0,C 180,E1 -27523.054,E2 -27523.054} C_VEL
LIN {X 0,Y 192.096,Z 666.388,A -85,B 0,C 180,E1 -27523.811,E2 -27523.811} C_VEL
LIN {X 0,Y 197.406,Z 651.986,A -85,B 0,C 180,E1 -27524.391,E2 -27524.391} C_VEL
LIN {X 0,Y 201.482,Z 637.256,A -85,B 0,C 180,E1 -27524.827,E2 -27524.827} C_VEL
LIN {X 0,Y 204.428,Z 621.455,A -85,B 0,C 180,E1 -27525.176,E2 -27525.176} C_VEL
LIN {X 0,Y 205.824,Z 610.785,A -85,B 0,C 180,E1 -27525.42,E2 -27525.42} C_VEL
LIN {X 0,Y 205.669,Z 609.422,A -85,B 0,C 180,E1 -27527.011,E2 -27527.011} C_VEL
LIN {X 0,Y 205.551,Z 609.116,A -85,B 0,C 180,E1 -27530.157,E2 -27530.157} C_VEL
LIN {X 0,Y 205.833,Z 609.561,A -85,B 0,C 180,E1 -27532.401,E2 -27532.401} C_VEL
LIN {X 0,Y 205.903,Z 610.096,A -85,B 0,C 180,E1 -27532.984,E2 -27532.984} C_VEL
LIN {X 0,Y 203.459,Z 627.283,A -85,B 0,C 180,E1 -27533.356,E2 -27533.356} C_VEL
LIN {X 0,Y 200.044,Z 642.469,A -85,B 0,C 180,E1 -27533.764,E2 -27533.764} C_VEL
LIN {X 0,Y 195.531,Z 656.891,A -85,B 0,C 180,E1 -27534.35,E2 -27534.35} C_VEL
LIN {X 0,Y 189.767,Z 671.064,A -85,B 0,C 180,E1 -27535.134,E2 -27535.134} C_VEL
LIN {X 0,Y 183.148,Z 684.172,A -85,B 0,C 180,E1 -27536.092,E2 -27536.092} C_VEL
LIN {X 0,Y 174.956,Z 697.548,A -85,B 0,C 180,E1 -27537.373,E2 -27537.373} C_VEL
LIN {X 0,Y 166.061,Z 709.671,A -85,B 0,C 180,E1 -27538.901,E2 -27538.901} C_VEL
LIN {X 0,Y 156.224,Z 721.05,A -85,B 0,C 180,E1 -27540.848,E2 -27540.848} C_VEL
LIN {X 0,Y 146.053,Z 731.139,A -85,B 0,C 180,E1 -27543.202,E2 -27543.202} C_VEL
LIN {X 0,Y 134.364,Z 741.027,A -85,B 0,C 180,E1 -27546.399,E2 -27546.399} C_VEL
LIN {X 0,Y 124.527,Z 748.165,A -85,B 0,C 180,E1 -27549.749,E2 -27549.749} C_VEL
LIN {X 0,Y 113.762,Z 754.933,A -85,B 0,C 180,E1 -27554.308,E2 -27554.308} C_VEL
LIN {X 0,Y 103.744,Z 760.321,A -85,B 0,C 180,E1 -27559.8,E2 -27559.8} C_VEL
LIN {X 0,Y 94.462,Z 764.558,A -85,B 0,C 180,E1 -27566.779,E2 -27566.779} C_VEL
LIN {X 0,Y 86.419,Z 767.562,A -85,B 0,C 180,E1 -27575.591,E2 -27575.591} C_VEL
LIN {X 0,Y 80.589,Z 769.133,A -85,B 0,C 180,E1 -27585.765,E2 -27585.765} C_VEL
LIN {X 0,Y 77.137,Z 769.332,A -85,B 0,C 180,E1 -27596.866,E2 -27596.866} C_VEL
LIN {X 0,Y 76.104,Z 768.207,A -85,B 0,C 180,E1 -27608.325,E2 -27608.325} C_VEL
LIN {X 0,Y 77.067,Z 765.814,A -85,B 0,C 180,E1 -27619.494,E2 -27619.494} C_VEL
LIN {X 0,Y 79.19,Z 763.185,A -85,B 0,C 180,E1 -27627.46,E2 -27627.46} C_VEL
LIN {X 0,Y 83.598,Z 758.496,A -85,B 0,C 180,E1 -27637.247,E2 -27637.247} C_VEL
LIN {X 0,Y 89.791,Z 752.383,A -85,B 0,C 180,E1 -27645.902,E2 -27645.902} C_VEL
LIN {X 0,Y 97.517,Z 744.676,A -85,B 0,C 180,E1 -27653.354,E2 -27653.354} C_VEL
LIN {X 0,Y 105.365,Z 736.382,A -85,B 0,C 180,E1 -27658.922,E2 -27658.922} C_VEL
LIN {X 0,Y 113.937,Z 726.426,A -85,B 0,C 180,E1 -27663.723,E2 -27663.723} C_VEL
LIN {X 0,Y 121.859,Z 716.195,A -85,B 0,C 180,E1 -27667.272,E2 -27667.272} C_VEL
LIN {X 0,Y 129.237,Z 705.408,A -85,B 0,C 180,E1 -27670.085,E2 -27670.085} C_VEL
LIN {X 0,Y 136.555,Z 693.142,A -85,B 0,C 180,E1 -27672.494,E2 -27672.494} C_VEL
LIN {X 0,Y 143.096,Z 680.238,A -85,B 0,C 180,E1 -27674.418,E2 -27674.418} C_VEL
LIN {X 0,Y 148.974,Z 666.181,A -85,B 0,C 180,E1 -27676.009,E2 -27676.009} C_VEL
LIN {X 0,Y 153.871,Z 651.565,A -85,B 0,C 180,E1 -27677.219,E2 -27677.219} C_VEL
LIN {X 0,Y 157.781,Z 636.058,A -85,B 0,C 180,E1 -27678.135,E2 -27678.135} C_VEL
LIN {X 0,Y 160.512,Z 620.301,A -85,B 0,C 180,E1 -27678.725,E2 -27678.725} C_VEL
LIN {X 0,Y 164.565,Z 583.11,A -85,B 0,C 180,E1 -27679.781,E2 -27679.781} C_VEL
LIN {X 0,Y 160.924,Z 574.79,A -85,B 0,C 180,E1 -27683.57,E2 -27683.57} C_VEL
LIN {X 0,Y 157.594,Z 567.873,A -85,B 0,C 180,E1 -27687.645,E2 -27687.645} C_VEL
LIN {X 0,Y 155.183,Z 563.221,A -85,B 0,C 180,E1 -27691.211,E2 -27691.211} C_VEL
LIN {X 0,Y 153.845,Z 560.711,A -85,B 0,C 180,E1 -27693.593,E2 -27693.593} C_VEL
LIN {X 0,Y 152.491,Z 558.012,A -85,B 0,C 180,E1 -27696.545,E2 -27696.545} C_VEL
LIN {X 0,Y 150.896,Z 554.733,A -85,B 0,C 180,E1 -27701.571,E2 -27701.571} C_VEL
LIN {X 0,Y 150.673,Z 554.187,A -85,B 0,C 180,E1 -27702.615,E2 -27702.615} C_VEL
LIN {X 0,Y 150.006,Z 553.402,A -85,B 0,C 180,E1 -27709.704,E2 -27709.704} C_VEL
LIN {X 0,Y 150.993,Z 554.202,A -85,B 0,C 180,E1 -27716.117,E2 -27716.117} C_VEL
LIN {X 0,Y 152.601,Z 557.643,A -85,B 0,C 180,E1 -27721.138,E2 -27721.138} C_VEL
LIN {X 0,Y 155.138,Z 562.762,A -85,B 0,C 180,E1 -27726.221,E2 -27726.221} C_VEL
LIN {X 0,Y 157.957,Z 568.514,A -85,B 0,C 180,E1 -27730.412,E2 -27730.412} C_VEL
LIN {X 0,Y 161.11,Z 575.132,A -85,B 0,C 180,E1 -27734.203,E2 -27734.203} C_VEL
LIN {X 0,Y 162.812,Z 579.341,A -85,B 0,C 180,E1 -27736.082,E2 -27736.082} C_VEL
LIN {X 0,Y 164.571,Z 585.095,A -85,B 0,C 180,E1 -27738.007,E2 -27738.007} C_VEL
LIN {X 0,Y 159.537,Z 629.453,A -85,B 0,C 180,E1 -27739.238,E2 -27739.238} C_VEL
LIN {X 0,Y 156.495,Z 644.899,A -85,B 0,C 180,E1 -27739.9,E2 -27739.9} C_VEL
LIN {X 0,Y 152.211,Z 659.921,A -85,B 0,C 180,E1 -27740.77,E2 -27740.77} C_VEL
LIN {X 0,Y 146.884,Z 674.541,A -85,B 0,C 180,E1 -27742.02,E2 -27742.02} C_VEL
LIN {X 0,Y 140.494,Z 688.604,A -85,B 0,C 180,E1 -27743.643,E2 -27743.643} C_VEL
LIN {X 0,Y 134.216,Z 700.22,A -85,B 0,C 180,E1 -27745.407,E2 -27745.407} C_VEL
LIN {X 0,Y 126.342,Z 712.797,A -85,B 0,C 180,E1 -27747.982,E2 -27747.982} C_VEL
LIN {X 0,Y 118.791,Z 723.337,A -85,B 0,C 180,E1 -27750.921,E2 -27750.921} C_VEL
LIN {X 0,Y 110.934,Z 733.091,A -85,B 0,C 180,E1 -27754.552,E2 -27754.552} C_VEL
LIN {X 0,Y 103.648,Z 741.408,A -85,B 0,C 180,E1 -27758.758,E2 -27758.758} C_VEL
LIN {X 0,Y 96.961,Z 748.528,A -85,B 0,C 180,E1 -27763.543,E2 -27763.543} C_VEL
LIN {X 0,Y 89.188,Z 756.326,A -85,B 0,C 180,E1 -27770.918,E2 -27770.918} C_VEL
LIN {X 0,Y 83.101,Z 762.5,A -85,B 0,C 180,E1 -27779.504,E2 -27779.504} C_VEL
LIN {X 0,Y 78.943,Z 767.214,A -85,B 0,C 180,E1 -27789.136,E2 -27789.136} C_VEL
LIN {X 0,Y 76.948,Z 770.584,A -85,B 0,C 180,E1 -27799.472,E2 -27799.472} C_VEL
LIN {X 0,Y 76.771,Z 772.688,A -85,B 0,C 180,E1 -27809.997,E2 -27809.997} C_VEL
LIN {X 0,Y 76.91,Z 773.557,A -85,B 0,C 180,E1 -27820.527,E2 -27820.527} C_VEL
LIN {X 0,Y 78.96,Z 773.329,A -85,B 0,C 180,E1 -27830.853,E2 -27830.853} C_VEL
LIN {X 0,Y 83.262,Z 771.966,A -85,B 0,C 180,E1 -27840.424,E2 -27840.424} C_VEL
LIN {X 0,Y 89.564,Z 769.498,A -85,B 0,C 180,E1 -27848.881,E2 -27848.881} C_VEL
LIN {X 0,Y 97.543,Z 765.906,A -85,B 0,C 180,E1 -27856.092,E2 -27856.092} C_VEL
LIN {X 0,Y 106.905,Z 761.101,A -85,B 0,C 180,E1 -27862.077,E2 -27862.077} C_VEL
LIN {X 0,Y 117.119,Z 754.98,A -85,B 0,C 180,E1 -27867.147,E2 -27867.147} C_VEL
LIN {X 0,Y 128.217,Z 747.379,A -85,B 0,C 180,E1 -27871.279,E2 -27871.279} C_VEL
LIN {X 0,Y 139.766,Z 738.186,A -85,B 0,C 180,E1 -27874.639,E2 -27874.639} C_VEL
LIN {X 0,Y 142.149,Z 735.947,A -85,B 0,C 180,E1 -27875.581,E2 -27875.581} C_VEL
LIN {X 0,Y 148.155,Z 729.004,A -85,B 0,C 180,E1 -27879.503,E2 -27879.503} C_VEL
LIN {X 0,Y 150.574,Z 726.469,A -85,B 0,C 180,E1 -27880.218,E2 -27880.218} C_VEL
LIN {X 0,Y 159.98,Z 716.464,A -85,B 0,C 180,E1 -27881.869,E2 -27881.869} C_VEL
LIN {X 0,Y 168.82,Z 705.559,A -85,B 0,C 180,E1 -27883.228,E2 -27883.228} C_VEL
LIN {X 0,Y 177.84,Z 692.411,A -85,B 0,C 180,E1 -27884.415,E2 -27884.415} C_VEL
LIN {X 0,Y 185.264,Z 679.399,A -85,B 0,C 180,E1 -27885.31,E2 -27885.31} C_VEL
LIN {X 0,Y 191.957,Z 665.102,A -85,B 0,C 180,E1 -27885.976,E2 -27885.976} C_VEL
LIN {X 0,Y 197.386,Z 650.297,A -85,B 0,C 180,E1 -27886.499,E2 -27886.499} C_VEL
LIN {X 0,Y 201.608,Z 634.67,A -85,B 0,C 180,E1 -27886.901,E2 -27886.901} C_VEL
LIN {X 0,Y 204.474,Z 618.232,A -85,B 0,C 180,E1 -27887.225,E2 -27887.225} C_VEL
LIN {X 0,Y 204.698,Z 616.415,A -85,B 0,C 180,E1 -27887.332,E2 -27887.332} C_VEL
LIN {X 0,Y 204.715,Z 616.249,A -85,B 0,C 180,E1 -27891.102,E2 -27891.102} C_VEL
LIN {X 0,Y 201.936,Z 632.875,A -85,B 0,C 180,E1 -27891.476,E2 -27891.476} C_VEL
LIN {X 0,Y 197.995,Z 647.986,A -85,B 0,C 180,E1 -27891.901,E2 -27891.901} C_VEL
LIN {X 0,Y 192.664,Z 662.964,A -85,B 0,C 180,E1 -27892.537,E2 -27892.537} C_VEL
LIN {X 0,Y 186.825,Z 675.823,A -85,B 0,C 180,E1 -27893.272,E2 -27893.272} C_VEL
LIN {X 0,Y 179.224,Z 689.522,A -85,B 0,C 180,E1 -27894.273,E2 -27894.273} C_VEL
LIN {X 0,Y 171.07,Z 701.749,A -85,B 0,C 180,E1 -27895.46,E2 -27895.46} C_VEL
LIN {X 0,Y 161.867,Z 713.404,A -85,B 0,C 180,E1 -27896.955,E2 -27896.955} C_VEL
LIN {X 0,Y 152.898,Z 723.154,A -85,B 0,C 180,E1 -27898.607,E2 -27898.607} C_VEL
LIN {X 0,Y 142.202,Z 733.152,A -85,B 0,C 180,E1 -27900.9,E2 -27900.9} C_VEL
LIN {X 0,Y 131.987,Z 741.372,A -85,B 0,C 180,E1 -27903.468,E2 -27903.468} C_VEL
LIN {X 0,Y 120.395,Z 749.388,A -85,B 0,C 180,E1 -27907.103,E2 -27907.103} C_VEL
LIN {X 0,Y 110.455,Z 755.252,A -85,B 0,C 180,E1 -27911.005,E2 -27911.005} C_VEL
LIN {X 0,Y 99.84,Z 760.601,A -85,B 0,C 180,E1 -27916.355,E2 -27916.355} C_VEL
LIN {X 0,Y 90.304,Z 764.627,A -85,B 0,C 180,E1 -27922.902,E2 -27922.902} C_VEL
LIN {X 0,Y 82.002,Z 767.497,A -85,B 0,C 180,E1 -27931.02,E2 -27931.02} C_VEL
LIN {X 0,Y 75.059,Z 769.238,A -85,B 0,C 180,E1 -27941.496,E2 -27941.496} C_VEL
LIN {X 0,Y 70.719,Z 769.601,A -85,B 0,C 180,E1 -27953.401,E2 -27953.401} C_VEL
LIN {X 0,Y 69.019,Z 768.579,A -85,B 0,C 180,E1 -27966.415,E2 -27966.415} C_VEL
LIN {X 0,Y 69.704,Z 766.409,A -85,B 0,C 180,E1 -27978.37,E2 -27978.37} C_VEL
LIN {X 0,Y 70.964,Z 764.808,A -85,B 0,C 180,E1 -27984.32,E2 -27984.32} C_VEL
LIN {X 0,Y 74.989,Z 760.633,A -85,B 0,C 180,E1 -27995.381,E2 -27995.381} C_VEL
LIN {X 0,Y 81.042,Z 755.066,A -85,B 0,C 180,E1 -28005.082,E2 -28005.082} C_VEL
LIN {X 0,Y 88.753,Z 747.968,A -85,B 0,C 180,E1 -28013.327,E2 -28013.327} C_VEL
LIN {X 0,Y 97.067,Z 739.91,A -85,B 0,C 180,E1 -28019.673,E2 -28019.673} C_VEL
LIN {X 0,Y 105.388,Z 731.111,A -85,B 0,C 180,E1 -28024.532,E2 -28024.532} C_VEL
LIN {X 0,Y 114.797,Z 719.997,A -85,B 0,C 180,E1 -28028.869,E2 -28028.869} C_VEL
LIN {X 0,Y 122.527,Z 709.608,A -85,B 0,C 180,E1 -28031.782,E2 -28031.782} C_VEL
LIN {X 0,Y 130.583,Z 697.141,A -85,B 0,C 180,E1 -28034.402,E2 -28034.402} C_VEL
LIN {X 0,Y 138.048,Z 683.517,A -85,B 0,C 180,E1 -28036.509,E2 -28036.509} C_VEL
LIN {X 0,Y 144.08,Z 670.161,A -85,B 0,C 180,E1 -28038.064,E2 -28038.064} C_VEL
LIN {X 0,Y 149.432,Z 655.534,A -85,B 0,C 180,E1 -28039.324,E2 -28039.324} C_VEL
LIN {X 0,Y 153.773,Z 639.998,A -85,B 0,C 180,E1 -28040.289,E2 -28040.289} C_VEL
LIN {X 0,Y 156.925,Z 624.035,A -85,B 0,C 180,E1 -28040.913,E2 -28040.913} C_VEL
LIN {X 0,Y 161.211,Z 586.502,A -85,B 0,C 180,E1 -28041.954,E2 -28041.954} C_VEL
LIN {X 0,Y 157.702,Z 578.338,A -85,B 0,C 180,E1 -28046.039,E2 -28046.039} C_VEL
LIN {X 0,Y 154.735,Z 571.951,A -85,B 0,C 180,E1 -28050.267,E2 -28050.267} C_VEL
LIN {X 0,Y 152.604,Z 567.619,A -85,B 0,C 180,E1 -28054.081,E2 -28054.081} C_VEL
LIN {X 0,Y 151.3,Z 564.869,A -85,B 0,C 180,E1 -28057.073,E2 -28057.073} C_VEL
LIN {X 0,Y 149.786,Z 561.445,A -85,B 0,C 180,E1 -28062.344,E2 -28062.344} C_VEL
LIN {X 0,Y 149.07,Z 560.435,A -85,B 0,C 180,E1 -28069.129,E2 -28069.129} C_VEL
LIN {X 0,Y 149.881,Z 561.014,A -85,B 0,C 180,E1 -28075.353,E2 -28075.353} C_VEL
LIN {X 0,Y 151.612,Z 565.037,A -85,B 0,C 180,E1 -28081.145,E2 -28081.145} C_VEL
LIN {X 0,Y 153.606,Z 569.266,A -85,B 0,C 180,E1 -28085.347,E2 -28085.347} C_VEL
LIN {X 0,Y 156.445,Z 575.491,A -85,B 0,C 180,E1 -28089.84,E2 -28089.84} C_VEL
LIN {X 0,Y 159.23,Z 581.735,A -85,B 0,C 180,E1 -28093.398,E2 -28093.398} C_VEL
LIN {X 0,Y 160.492,Z 585.355,A -85,B 0,C 180,E1 -28094.907,E2 -28094.907} C_VEL
LIN {X 0,Y 161.209,Z 587.829,A -85,B 0,C 180,E1 -28095.783,E2 -28095.783} C_VEL
LIN {X 0,Y 156.496,Z 628.672,A -85,B 0,C 180,E1 -28096.891,E2 -28096.891} C_VEL
LIN {X 0,Y 153.4,Z 644.311,A -85,B 0,C 180,E1 -28097.535,E2 -28097.535} C_VEL
LIN {X 0,Y 149.021,Z 659.428,A -85,B 0,C 180,E1 -28098.354,E2 -28098.354} C_VEL
LIN {X 0,Y 143.567,Z 674.117,A -85,B 0,C 180,E1 -28099.549,E2 -28099.549} C_VEL
LIN {X 0,Y 136.852,Z 688.506,A -85,B 0,C 180,E1 -28101.132,E2 -28101.132} C_VEL
LIN {X 0,Y 130.542,Z 699.855,A -85,B 0,C 180,E1 -28102.783,E2 -28102.783} C_VEL
LIN {X 0,Y 122.399,Z 712.459,A -85,B 0,C 180,E1 -28105.262,E2 -28105.262} C_VEL
LIN {X 0,Y 113.861,Z 723.93,A -85,B 0,C 180,E1 -28108.407,E2 -28108.407} C_VEL
LIN {X 0,Y 104.79,Z 734.562,A -85,B 0,C 180,E1 -28112.447,E2 -28112.447} C_VEL
LIN {X 0,Y 95.688,Z 744.268,A -85,B 0,C 180,E1 -28117.853,E2 -28117.853} C_VEL
LIN {X 0,Y 87.781,Z 751.879,A -85,B 0,C 180,E1 -28123.896,E2 -28123.896} C_VEL
LIN {X 0,Y 79.996,Z 759.052,A -85,B 0,C 180,E1 -28132.248,E2 -28132.248} C_VEL
LIN {X 0,Y 74.401,Z 764.477,A -85,B 0,C 180,E1 -28141.813,E2 -28141.813} C_VEL
LIN {X 0,Y 70.813,Z 768.599,A -85,B 0,C 180,E1 -28152.675,E2 -28152.675} C_VEL
LIN {X 0,Y 69.56,Z 771.423,A -85,B 0,C 180,E1 -28164.198,E2 -28164.198} C_VEL
LIN {X 0,Y 69.69,Z 772.369,A -85,B 0,C 180,E1 -28169.997,E2 -28169.997} C_VEL
LIN {X 0,Y 69.918,Z 773.326,A -85,B 0,C 180,E1 -28181.594,E2 -28181.594} C_VEL
LIN {X 0,Y 72.311,Z 773.171,A -85,B 0,C 180,E1 -28192.874,E2 -28192.874} C_VEL
LIN {X 0,Y 77.166,Z 771.877,A -85,B 0,C 180,E1 -28203.121,E2 -28203.121} C_VEL
LIN {X 0,Y 84.105,Z 769.508,A -85,B 0,C 180,E1 -28211.947,E2 -28211.947} C_VEL
LIN {X 0,Y 92.72,Z 766.018,A -85,B 0,C 180,E1 -28219.282,E2 -28219.282} C_VEL
LIN {X 0,Y 102.686,Z 761.339,A -85,B 0,C 180,E1 -28225.21,E2 -28225.21} C_VEL
LIN {X 0,Y 113.406,Z 755.328,A -85,B 0,C 180,E1 -28230.177,E2 -28230.177} C_VEL
LIN {X 0,Y 124.972,Z 747.843,A -85,B 0,C 180,E1 -28234.125,E2 -28234.125} C_VEL
LIN {X 0,Y 137.065,Z 738.695,A -85,B 0,C 180,E1 -28237.355,E2 -28237.355} C_VEL
LIN {X 0,Y 147.968,Z 729.034,A -85,B 0,C 180,E1 -28239.722,E2 -28239.722} C_VEL
LIN {X 0,Y 150.574,Z 726.469,A -85,B 0,C 180,E1 -28240.218,E2 -28240.218} C_VEL
LIN {X 0,Y 154.322,Z 722.581,A -85,B 0,C 180,E1 -28241.11,E2 -28241.11} C_VEL
LIN {X 0,Y 164.804,Z 709.666,A -85,B 0,C 180,E1 -28244.982,E2 -28244.982} C_VEL
LIN {X 0,Y 168.198,Z 705.271,A -85,B 0,C 180,E1 -28245.681,E2 -28245.681} C_VEL
LIN {X 0,Y 176.934,Z 692.83,A -85,B 0,C 180,E1 -28246.688,E2 -28246.688} C_VEL
LIN {X 0,Y 184.468,Z 679.956,A -85,B 0,C 180,E1 -28247.488,E2 -28247.488} C_VEL
LIN {X 0,Y 190.392,Z 667.767,A -85,B 0,C 180,E1 -28248.007,E2 -28248.007} C_VEL
LIN {X 0,Y 196.175,Z 652.959,A -85,B 0,C 180,E1 -28248.492,E2 -28248.492} C_VEL
LIN {X 0,Y 200.723,Z 637.327,A -85,B 0,C 180,E1 -28248.871,E2 -28248.871} C_VEL
LIN {X 0,Y 203.547,Z 623.227,A -85,B 0,C 180,E1 -28249.16,E2 -28249.16} C_VEL
LIN {X 0,Y 203.546,Z 623.222,A -85,B 0,C 180,E1 -28249.234,E2 -28249.234} C_VEL
LIN {X 0,Y 200.446,Z 638.386,A -85,B 0,C 180,E1 -28249.586,E2 -28249.586} C_VEL
LIN {X 0,Y 196.176,Z 652.843,A -85,B 0,C 180,E1 -28249.997,E2 -28249.997} C_VEL
LIN {X 0,Y 190.549,Z 667.241,A -85,B 0,C 180,E1 -28250.605,E2 -28250.605} C_VEL
LIN {X 0,Y 183.726,Z 681.069,A -85,B 0,C 180,E1 -28251.393,E2 -28251.393} C_VEL
LIN {X 0,Y 175.59,Z 694.5,A -85,B 0,C 180,E1 -28252.377,E2 -28252.377} C_VEL
LIN {X 0,Y 166.176,Z 707.354,A -85,B 0,C 180,E1 -28253.635,E2 -28253.635} C_VEL
LIN {X 0,Y 157.005,Z 717.946,A -85,B 0,C 180,E1 -28255.033,E2 -28255.033} C_VEL
LIN {X 0,Y 147.838,Z 727.146,A -85,B 0,C 180,E1 -28256.629,E2 -28256.629} C_VEL
LIN {X 0,Y 137.071,Z 736.4,A -85,B 0,C 180,E1 -28258.794,E2 -28258.794} C_VEL
LIN {X 0,Y 124.805,Z 745.369,A -85,B 0,C 180,E1 -28261.825,E2 -28261.825} C_VEL
LIN {X 0,Y 112.965,Z 752.647,A -85,B 0,C 180,E1 -28265.51,E2 -28265.51} C_VEL
LIN {X 0,Y 103.257,Z 757.706,A -85,B 0,C 180,E1 -28269.296,E2 -28269.296} C_VEL
LIN {X 0,Y 94.096,Z 761.86,A -85,B 0,C 180,E1 -28273.853,E2 -28273.853} C_VEL
LIN {X 0,Y 83.034,Z 765.951,A -85,B 0,C 180,E1 -28281.412,E2 -28281.412} C_VEL
LIN {X 0,Y 73.776,Z 768.564,A -85,B 0,C 180,E1 -28290.986,E2 -28290.986} C_VEL
LIN {X 0,Y 66.911,Z 769.778,A -85,B 0,C 180,E1 -28302.678,E2 -28302.678} C_VEL
LIN {X 0,Y 62.908,Z 769.633,A -85,B 0,C 180,E1 -28316.046,E2 -28316.046} C_VEL
LIN {X 0,Y 61.957,Z 768.801,A -85,B 0,C 180,E1 -28325.162,E2 -28325.162} C_VEL
LIN {X 0,Y 62.375,Z 766.96,A -85,B 0,C 180,E1 -28336.981,E2 -28336.981} C_VEL
LIN {X 0,Y 65.343,Z 763.572,A -85,B 0,C 180,E1 -28350.003,E2 -28350.003} C_VEL
LIN {X 0,Y 70.602,Z 758.867,A -85,B 0,C 180,E1 -28361.487,E2 -28361.487} C_VEL
LIN {X 0,Y 77.881,Z 752.739,A -85,B 0,C 180,E1 -28371.162,E2 -28371.162} C_VEL
LIN {X 0,Y 86.728,Z 745.018,A -85,B 0,C 180,E1 -28379.094,E2 -28379.094} C_VEL
LIN {X 0,Y 95.553,Z 736.693,A -85,B 0,C 180,E1 -28384.764,E2 -28384.764} C_VEL
LIN {X 0,Y 104.989,Z 726.727,A -85,B 0,C 180,E1 -28389.492,E2 -28389.492} C_VEL
LIN {X 0,Y 113.592,Z 716.473,A -85,B 0,C 180,E1 -28392.891,E2 -28392.891} C_VEL
LIN {X 0,Y 122.517,Z 704.254,A -85,B 0,C 180,E1 -28395.813,E2 -28395.813} C_VEL
LIN {X 0,Y 130.107,Z 692.042,A -85,B 0,C 180,E1 -28397.967,E2 -28397.967} C_VEL
LIN {X 0,Y 137.058,Z 678.8,A -85,B 0,C 180,E1 -28399.709,E2 -28399.709} C_VEL
LIN {X 0,Y 142.91,Z 665.254,A -85,B 0,C 180,E1 -28401.045,E2 -28401.045} C_VEL
LIN {X 0,Y 148.01,Z 650.384,A -85,B 0,C 180,E1 -28402.132,E2 -28402.132} C_VEL
LIN {X 0,Y 151.896,Z 635.231,A -85,B 0,C 180,E1 -28402.919,E2 -28402.919} C_VEL
LIN {X 0,Y 154.566,Z 620.017,A -85,B 0,C 180,E1 -28403.422,E2 -28403.422} C_VEL
LIN {X 0,Y 157.991,Z 590.04,A -85,B 0,C 180,E1 -28404.231,E2 -28404.231} C_VEL
LIN {X 0,Y 155.18,Z 583.049,A -85,B 0,C 180,E1 -28407.982,E2 -28407.982} C_VEL
LIN {X 0,Y 152.431,Z 576.896,A -85,B 0,C 180,E1 -28412.423,E2 -28412.423} C_VEL
LIN {X 0,Y 151.017,Z 573.79,A -85,B 0,C 180,E1 -28415.371,E2 -28415.371} C_VEL
LIN {X 0,Y 149.927,Z 571.459,A -85,B 0,C 180,E1 -28418.117,E2 -28418.117} C_VEL
LIN {X 0,Y 148.605,Z 568.143,A -85,B 0,C 180,E1 -28423.515,E2 -28423.515} C_VEL
LIN {X 0,Y 148.141,Z 567.484,A -85,B 0,C 180,E1 -28429.06,E2 -28429.06} C_VEL
LIN {X 0,Y 148.885,Z 568.086,A -85,B 0,C 180,E1 -28435.137,E2 -28435.137} C_VEL
LIN {X 0,Y 150.397,Z 571.906,A -85,B 0,C 180,E1 -28440.577,E2 -28440.577} C_VEL
LIN {X 0,Y 152.257,Z 576.167,A -85,B 0,C 180,E1 -28444.757,E2 -28444.757} C_VEL
LIN {X 0,Y 155.024,Z 582.599,A -85,B 0,C 180,E1 -28449.361,E2 -28449.361} C_VEL
LIN {X 0,Y 157.615,Z 589.066,A -85,B 0,C 180,E1 -28452.882,E2 -28452.882} C_VEL
LIN {X 0,Y 158.066,Z 590.733,A -85,B 0,C 180,E1 -28453.498,E2 -28453.498} C_VEL
LIN {X 0,Y 153.686,Z 628.032,A -85,B 0,C 180,E1 -28454.486,E2 -28454.486} C_VEL
LIN {X 0,Y 150.378,Z 644.372,A -85,B 0,C 180,E1 -28455.117,E2 -28455.117} C_VEL
LIN {X 0,Y 146.114,Z 658.855,A -85,B 0,C 180,E1 -28455.845,E2 -28455.845} C_VEL
LIN {X 0,Y 140.523,Z 673.621,A -85,B 0,C 180,E1 -28456.958,E2 -28456.958} C_VEL
LIN {X 0,Y 134.176,Z 687.056,A -85,B 0,C 180,E1 -28458.316,E2 -28458.316} C_VEL
LIN {X 0,Y 127.956,Z 698.156,A -85,B 0,C 180,E1 -28459.846,E2 -28459.846} C_VEL
LIN {X 0,Y 121.067,Z 708.853,A -85,B 0,C 180,E1 -28461.747,E2 -28461.747} C_VEL
LIN {X 0,Y 113.56,Z 719.053,A -85,B 0,C 180,E1 -28464.095,E2 -28464.095} C_VEL
LIN {X 0,Y 104.85,Z 729.429,A -85,B 0,C 180,E1 -28467.357,E2 -28467.357} C_VEL
LIN {X 0,Y 95.283,Z 739.566,A -85,B 0,C 180,E1 -28471.976,E2 -28471.976} C_VEL
LIN {X 0,Y 86.462,Z 747.971,A -85,B 0,C 180,E1 -28477.575,E2 -28477.575} C_VEL
LIN {X 0,Y 78.558,Z 754.889,A -85,B 0,C 180,E1 -28484.296,E2 -28484.296} C_VEL
LIN {X 0,Y 71.104,Z 761.278,A -85,B 0,C 180,E1 -28493.623,E2 -28493.623} C_VEL
LIN {X 0,Y 65.752,Z 766.189,A -85,B 0,C 180,E1 -28504.685,E2 -28504.685} C_VEL
LIN {X 0,Y 62.953,Z 769.754,A -85,B 0,C 180,E1 -28517.095,E2 -28517.095} C_VEL
LIN {X 0,Y 62.598,Z 772.047,A -85,B 0,C 180,E1 -28529.996,E2 -28529.996} C_VEL
LIN {X 0,Y 62.931,Z 773.093,A -85,B 0,C 180,E1 -28542.902,E2 -28542.902} C_VEL
LIN {X 0,Y 65.771,Z 772.986,A -85,B 0,C 180,E1 -28555.3,E2 -28555.3} C_VEL
LIN {X 0,Y 71.273,Z 771.788,A -85,B 0,C 180,E1 -28566.269,E2 -28566.269} C_VEL
LIN {X 0,Y 78.922,Z 769.524,A -85,B 0,C 180,E1 -28575.426,E2 -28575.426} C_VEL
LIN {X 0,Y 88.226,Z 766.155,A -85,B 0,C 180,E1 -28582.801,E2 -28582.801} C_VEL
LIN {X 0,Y 98.789,Z 761.552,A -85,B 0,C 180,E1 -28588.61,E2 -28588.61} C_VEL
LIN {X 0,Y 110.367,Z 755.458,A -85,B 0,C 180,E1 -28593.53,E2 -28593.53} C_VEL
LIN {X 0,Y 123.591,Z 747.32,A -85,B 0,C 180,E1 -28597.52,E2 -28597.52} C_VEL
LIN {X 0,Y 136.098,Z 738.113,A -85,B 0,C 180,E1 -28600.454,E2 -28600.454} C_VEL
LIN {X 0,Y 147.281,Z 728.398,A -85,B 0,C 180,E1 -28602.617,E2 -28602.617} C_VEL
LIN {X 0,Y 158.516,Z 716.934,A -85,B 0,C 180,E1 -28604.368,E2 -28604.368} C_VEL
LIN {X 0,Y 168.198,Z 705.271,A -85,B 0,C 180,E1 -28605.681,E2 -28605.681} C_VEL
LIN {X 0,Y 170.408,Z 702.301,A -85,B 0,C 180,E1 -28606.19,E2 -28606.19} C_VEL
LIN {X 0,Y 176.458,Z 693.116,A -85,B 0,C 180,E1 -28608.776,E2 -28608.776} C_VEL
LIN {X 0,Y 178.439,Z 689.913,A -85,B 0,C 180,E1 -28609.194,E2 -28609.194} C_VEL
LIN {X 0,Y 178.842,Z 689.257,A -85,B 0,C 180,E1 -28609.234,E2 -28609.234} C_VEL
LIN {X 0,Y 178.587,Z 689.642,A -85,B 0,C 180,E1 -28609.673,E2 -28609.673} C_VEL
LIN {X 0,Y 169.902,Z 702.232,A -85,B 0,C 180,E1 -28610.66,E2 -28610.66} C_VEL
LIN {X 0,Y 160.734,Z 713.415,A -85,B 0,C 180,E1 -28611.802,E2 -28611.802} C_VEL
LIN {X 0,Y 150.37,Z 724.159,A -85,B 0,C 180,E1 -28613.286,E2 -28613.286} C_VEL
LIN {X 0,Y 139.294,Z 733.914,A -85,B 0,C 180,E1 -28615.158,E2 -28615.158} C_VEL
LIN {X 0,Y 128.459,Z 742.081,A -85,B 0,C 180,E1 -28617.309,E2 -28617.309} C_VEL
LIN {X 0,Y 117.589,Z 749.104,A -85,B 0,C 180,E1 -28620.001,E2 -28620.001} C_VEL
LIN {X 0,Y 105.116,Z 755.889,A -85,B 0,C 180,E1 -28623.835,E2 -28623.835} C_VEL
LIN {X 0,Y 92.5,Z 761.51,A -85,B 0,C 180,E1 -28629.007,E2 -28629.007} C_VEL
LIN {X 0,Y 80.447,Z 765.782,A -85,B 0,C 180,E1 -28636.072,E2 -28636.072} C_VEL
LIN {X 0,Y 69.998,Z 768.559,A -85,B 0,C 180,E1 -28645.369,E2 -28645.369} C_VEL
LIN {X 0,Y 61.796,Z 769.919,A -85,B 0,C 180,E1 -28657.247,E2 -28657.247} C_VEL
LIN {X 0,Y 56.575,Z 769.916,A -85,B 0,C 180,E1 -28671.607,E2 -28671.607} C_VEL
LIN {X 0,Y 54.776,Z 768.596,A -85,B 0,C 180,E1 -28687.366,E2 -28687.366} C_VEL
LIN {X 0,Y 56.114,Z 766.003,A -85,B 0,C 180,E1 -28702.809,E2 -28702.809} C_VEL
LIN {X 0,Y 60.383,Z 762.12,A -85,B 0,C 180,E1 -28716.687,E2 -28716.687} C_VEL
LIN {X 0,Y 67.04,Z 756.888,A -85,B 0,C 180,E1 -28728.334,E2 -28728.334} C_VEL
LIN {X 0,Y 75.625,Z 750.167,A -85,B 0,C 180,E1 -28737.691,E2 -28737.691} C_VEL
LIN {X 0,Y 84.315,Z 742.902,A -85,B 0,C 180,E1 -28744.241,E2 -28744.241} C_VEL
LIN {X 0,Y 93.835,Z 734.133,A -85,B 0,C 180,E1 -28749.543,E2 -28749.543} C_VEL
LIN {X 0,Y 103.91,Z 723.572,A -85,B 0,C 180,E1 -28753.891,E2 -28753.891} C_VEL
LIN {X 0,Y 113.149,Z 712.491,A -85,B 0,C 180,E1 -28757.006,E2 -28757.006} C_VEL
LIN {X 0,Y 122.257,Z 699.648,A -85,B 0,C 180,E1 -28759.615,E2 -28759.615} C_VEL
LIN {X 0,Y 130.145,Z 686.457,A -85,B 0,C 180,E1 -28761.54,E2 -28761.54} C_VEL
LIN {X 0,Y 136.489,Z 673.687,A -85,B 0,C 180,E1 -28762.952,E2 -28762.952} C_VEL
LIN {X 0,Y 142.496,Z 658.777,A -85,B 0,C 180,E1 -28764.167,E2 -28764.167} C_VEL
LIN {X 0,Y 147.343,Z 643.057,A -85,B 0,C 180,E1 -28765.083,E2 -28765.083} C_VEL
LIN {X 0,Y 150.701,Z 627.836,A -85,B 0,C 180,E1 -28765.679,E2 -28765.679} C_VEL
LIN {X 0,Y 153.543,Z 606.778,A -85,B 0,C 180,E1 -28766.212,E2 -28766.212} C_VEL
LIN {X 0,Y 155.038,Z 593.739,A -85,B 0,C 180,E1 -28766.547,E2 -28766.547} C_VEL
LIN {X 0,Y 152.734,Z 587.804,A -85,B 0,C 180,E1 -28770.047,E2 -28770.047} C_VEL
LIN {X 0,Y 150.551,Z 582.464,A -85,B 0,C 180,E1 -28774.159,E2 -28774.159} C_VEL
LIN {X 0,Y 148.825,Z 578.391,A -85,B 0,C 180,E1 -28778.523,E2 -28778.523} C_VEL
LIN {X 0,Y 147.691,Z 575.235,A -85,B 0,C 180,E1 -28783.41,E2 -28783.41} C_VEL
LIN {X 0,Y 147.215,Z 574.507,A -85,B 0,C 180,E1 -28788.991,E2 -28788.991} C_VEL
LIN {X 0,Y 147.814,Z 575.002,A -85,B 0,C 180,E1 -28794.543,E2 -28794.543} C_VEL
LIN {X 0,Y 149.133,Z 578.648,A -85,B 0,C 180,E1 -28799.826,E2 -28799.826} C_VEL
LIN {X 0,Y 150.643,Z 582.345,A -85,B 0,C 180,E1 -28803.552,E2 -28803.552} C_VEL
LIN {X 0,Y 152.994,Z 588.277,A -85,B 0,C 180,E1 -28807.92,E2 -28807.92} C_VEL
LIN {X 0,Y 155.133,Z 593.959,A -85,B 0,C 180,E1 -28811.162,E2 -28811.162} C_VEL
LIN {X 0,Y 151.133,Z 627.265,A -85,B 0,C 180,E1 -28812.009,E2 -28812.009} C_VEL
LIN {X 0,Y 147.964,Z 643.001,A -85,B 0,C 180,E1 -28812.551,E2 -28812.551} C_VEL
LIN {X 0,Y 143.494,Z 658.13,A -85,B 0,C 180,E1 -28813.234,E2 -28813.234} C_VEL
LIN {X 0,Y 137.779,Z 673.023,A -85,B 0,C 180,E1 -28814.26,E2 -28814.26} C_VEL
LIN {X 0,Y 131.296,Z 686.513,A -85,B 0,C 180,E1 -28815.523,E2 -28815.523} C_VEL
LIN {X 0,Y 124.086,Z 698.962,A -85,B 0,C 180,E1 -28817.101,E2 -28817.101} C_VEL
LIN {X 0,Y 115.424,Z 711.648,A -85,B 0,C 180,E1 -28819.301,E2 -28819.301} C_VEL
LIN {X 0,Y 106.248,Z 723.189,A -85,B 0,C 180,E1 -28822.167,E2 -28822.167} C_VEL
LIN {X 0,Y 96.324,Z 733.941,A -85,B 0,C 180,E1 -28825.961,E2 -28825.961} C_VEL
LIN {X 0,Y 86.239,Z 743.642,A -85,B 0,C 180,E1 -28831.16,E2 -28831.16} C_VEL
LIN {X 0,Y 77.253,Z 751.284,A -85,B 0,C 180,E1 -28837.244,E2 -28837.244} C_VEL
LIN {X 0,Y 68.069,Z 758.577,A -85,B 0,C 180,E1 -28846.279,E2 -28846.279} C_VEL
LIN {X 0,Y 62.118,Z 763.322,A -85,B 0,C 180,E1 -28855.545,E2 -28855.545} C_VEL
LIN {X 0,Y 57.326,Z 767.653,A -85,B 0,C 180,E1 -28868.417,E2 -28868.417} C_VEL
LIN {X 0,Y 55.428,Z 770.676,A -85,B 0,C 180,E1 -28882.712,E2 -28882.712} C_VEL
LIN {X 0,Y 55.495,Z 771.718,A -85,B 0,C 180,E1 -28889.996,E2 -28889.996} C_VEL
LIN {X 0,Y 55.998,Z 772.84,A -85,B 0,C 180,E1 -28904.533,E2 -28904.533} C_VEL
LIN {X 0,Y 59.378,Z 772.8,A -85,B 0,C 180,E1 -28918.253,E2 -28918.253} C_VEL
LIN {X 0,Y 65.636,Z 771.707,A -85,B 0,C 180,E1 -28929.97,E2 -28929.97} C_VEL
LIN {X 0,Y 74.069,Z 769.551,A -85,B 0,C 180,E1 -28939.377,E2 -28939.377} C_VEL
LIN {X 0,Y 84.102,Z 766.264,A -85,B 0,C 180,E1 -28946.678,E2 -28946.678} C_VEL
LIN {X 0,Y 95.265,Z 761.758,A -85,B 0,C 180,E1 -28952.28,E2 -28952.28} C_VEL
LIN {X 0,Y 107.026,Z 755.999,A -85,B 0,C 180,E1 -28956.821,E2 -28956.821} C_VEL
LIN {X 0,Y 119.468,Z 748.807,A -85,B 0,C 180,E1 -28960.254,E2 -28960.254} C_VEL
LIN {X 0,Y 132.274,Z 739.983,A -85,B 0,C 180,E1 -28963.006,E2 -28963.006} C_VEL
LIN {X 0,Y 143.7,Z 730.704,A -85,B 0,C 180,E1 -28964.99,E2 -28964.99} C_VEL
LIN {X 0,Y 155.037,Z 719.865,A -85,B 0,C 180,E1 -28966.609,E2 -28966.609} C_VEL
LIN {X 0,Y 165.337,Z 708.217,A -85,B 0,C 180,E1 -28967.857,E2 -28967.857} C_VEL
LIN {X 0,Y 173.77,Z 697.011,A -85,B 0,C 180,E1 -28968.736,E2 -28968.736} C_VEL
LIN {X 0,Y 178.439,Z 689.913,A -85,B 0,C 180,E1 -28969.194,E2 -28969.194} C_VEL
LIN {X 0,Y 177.314,Z 691.705,A -85,B 0,C 180,E1 -28969.459,E2 -28969.459} C_VEL
LIN {X 0,Y 173.886,Z 696.77,A -85,B 0,C 180,E1 -28969.635,E2 -28969.635} C_VEL
LIN {X 0,Y 166.132,Z 707.028,A -85,B 0,C 180,E1 -28969.616,E2 -28969.616} C_VEL
LIN {X 0,Y 160.899,Z 713.183,A -85,B 0,C 180,E1 -28969.49,E2 -28969.49} C_VEL
LIN {X 0,Y 155.477,Z 719.039,A -85,B 0,C 180,E1 -28969.222,E2 -28969.222} C_VEL
LIN {X 0,Y 149.845,Z 724.584,A -85,B 0,C 180,E1 -28968.727,E2 -28968.727} C_VEL
LIN {X 0,Y 140.386,Z 733.019,A -85,B 0,C 180,E1 -28967.466,E2 -28967.466} C_VEL
LIN {X 0,Y 128.738,Z 741.889,A -85,B 0,C 180,E1 -28965.687,E2 -28965.687} C_VEL
LIN {X 0,Y 117.265,Z 749.317,A -85,B 0,C 180,E1 -28963.511,E2 -28963.511} C_VEL
LIN {X 0,Y 103.625,Z 756.762,A -85,B 0,C 180,E1 -28960.179,E2 -28960.179} C_VEL
LIN {X 0,Y 92.163,Z 761.983,A -85,B 0,C 180,E1 -28956.209,E2 -28956.209} C_VEL
LIN {X 0,Y 80.395,Z 766.361,A -85,B 0,C 180,E1 -28950.942,E2 -28950.942} C_VEL
LIN {X 0,Y 69.623,Z 769.574,A -85,B 0,C 180,E1 -28943.851,E2 -28943.851} C_VEL
LIN {X 0,Y 60.327,Z 771.628,A -85,B 0,C 180,E1 -28934.34,E2 -28934.34} C_VEL
LIN {X 0,Y 53.188,Z 772.617,A -85,B 0,C 180,E1 -28921.902,E2 -28921.902} C_VEL
LIN {X 0,Y 49.134,Z 772.556,A -85,B 0,C 180,E1 -28906.618,E2 -28906.618} C_VEL
LIN {X 0,Y 48.381,Z 771.388,A -85,B 0,C 180,E1 -28889.995,E2 -28889.995} C_VEL
LIN {X 0,Y 49.146,Z 768.895,A -85,B 0,C 180,E1 -28873.377,E2 -28873.377} C_VEL
LIN {X 0,Y 53.167,Z 765.12,A -85,B 0,C 180,E1 -28858.075,E2 -28858.075} C_VEL
LIN {X 0,Y 60.118,Z 759.984,A -85,B 0,C 180,E1 -28845.454,E2 -28845.454} C_VEL
LIN {X 0,Y 69.285,Z 753.36,A -85,B 0,C 180,E1 -28835.754,E2 -28835.754} C_VEL
LIN {X 0,Y 78.545,Z 746.186,A -85,B 0,C 180,E1 -28829.256,E2 -28829.256} C_VEL
LIN {X 0,Y 88.475,Z 737.484,A -85,B 0,C 180,E1 -28824.002,E2 -28824.002} C_VEL
LIN {X 0,Y 97.523,Z 728.671,A -85,B 0,C 180,E1 -28820.466,E2 -28820.466} C_VEL
LIN {X 0,Y 106.892,Z 718.248,A -85,B 0,C 180,E1 -28817.564,E2 -28817.564} C_VEL
LIN {X 0,Y 116.488,Z 705.755,A -85,B 0,C 180,E1 -28815.13,E2 -28815.13} C_VEL
LIN {X 0,Y 122.184,Z 697.191,A -85,B 0,C 180,E1 -28813.912,E2 -28813.912} C_VEL
LIN {X 0,Y 129.559,Z 684.373,A -85,B 0,C 180,E1 -28812.462,E2 -28812.462} C_VEL
LIN {X 0,Y 135.353,Z 672.405,A -85,B 0,C 180,E1 -28811.457,E2 -28811.457} C_VEL
LIN {X 0,Y 141.184,Z 657.373,A -85,B 0,C 180,E1 -28810.533,E2 -28810.533} C_VEL
LIN {X 0,Y 145.552,Z 642.792,A -85,B 0,C 180,E1 -28809.95,E2 -28809.95} C_VEL
LIN {X 0,Y 148.812,Z 626.755,A -85,B 0,C 180,E1 -28809.435,E2 -28809.435} C_VEL
LIN {X 0,Y 152.391,Z 597.7,A -85,B 0,C 180,E1 -28808.736,E2 -28808.736} C_VEL
LIN {X 0,Y 150.242,Z 591.814,A -85,B 0,C 180,E1 -28804.924,E2 -28804.924} C_VEL
LIN {X 0,Y 148.744,Z 587.565,A -85,B 0,C 180,E1 -28801.447,E2 -28801.447} C_VEL
LIN {X 0,Y 147.569,Z 584.511,A -85,B 0,C 180,E1 -28797.939,E2 -28797.939} C_VEL
LIN {X 0,Y 146.75,Z 581.958,A -85,B 0,C 180,E1 -28793.921,E2 -28793.921} C_VEL
LIN {X 0,Y 146.288,Z 581.542,A -85,B 0,C 180,E1 -28788.92,E2 -28788.92} C_VEL
LIN {X 0,Y 146.692,Z 582.336,A -85,B 0,C 180,E1 -28783.68,E2 -28783.68} C_VEL
LIN {X 0,Y 148.002,Z 586.132,A -85,B 0,C 180,E1 -28778.036,E2 -28778.036} C_VEL
LIN {X 0,Y 149.42,Z 589.742,A -85,B 0,C 180,E1 -28774.41,E2 -28774.41} C_VEL
LIN {X 0,Y 151.616,Z 595.605,A -85,B 0,C 180,E1 -28770.102,E2 -28770.102} C_VEL
LIN {X 0,Y 152.296,Z 597.503,A -85,B 0,C 180,E1 -28768.977,E2 -28768.977} C_VEL
LIN {X 0,Y 148.858,Z 625.121,A -85,B 0,C 180,E1 -28768.298,E2 -28768.298} C_VEL
LIN {X 0,Y 145.545,Z 640.757,A -85,B 0,C 180,E1 -28767.814,E2 -28767.814} C_VEL
LIN {X 0,Y 140.877,Z 656.368,A -85,B 0,C 180,E1 -28767.008,E2 -28767.008} C_VEL
LIN {X 0,Y 135.548,Z 670.055,A -85,B 0,C 180,E1 -28766.058,E2 -28766.058} C_VEL
LIN {X 0,Y 129.042,Z 683.527,A -85,B 0,C 180,E1 -28764.782,E2 -28764.782} C_VEL
LIN {X 0,Y 120.921,Z 697.287,A -85,B 0,C 180,E1 -28763.052,E2 -28763.052} C_VEL
LIN {X 0,Y 112.082,Z 709.823,A -85,B 0,C 180,E1 -28760.854,E2 -28760.854} C_VEL
LIN {X 0,Y 101.939,Z 721.976,A -85,B 0,C 180,E1 -28757.831,E2 -28757.831} C_VEL
LIN {X 0,Y 92.788,Z 731.464,A -85,B 0,C 180,E1 -28754.479,E2 -28754.479} C_VEL
LIN {X 0,Y 83.373,Z 740.047,A -85,B 0,C 180,E1 -28750.071,E2 -28750.071} C_VEL
LIN {X 0,Y 73.089,Z 748.395,A -85,B 0,C 180,E1 -28743.569,E2 -28743.569} C_VEL
LIN {X 0,Y 64.5,Z 754.705,A -85,B 0,C 180,E1 -28735.843,E2 -28735.843} C_VEL
LIN {X 0,Y 56.308,Z 760.488,A -85,B 0,C 180,E1 -28724.459,E2 -28724.459} C_VEL
LIN {X 0,Y 50.486,Z 764.873,A -85,B 0,C 180,E1 -28710.004,E2 -28710.004} C_VEL
LIN {X 0,Y 47.754,Z 767.954,A -85,B 0,C 180,E1 -28692.887,E2 -28692.887} C_VEL
LIN {X 0,Y 47.917,Z 769.23,A -85,B 0,C 180,E1 -28681.65,E2 -28681.65} C_VEL
LIN {X 0,Y 51.709,Z 770.275,A -85,B 0,C 180,E1 -28662.813,E2 -28662.813} C_VEL
LIN {X 0,Y 58.79,Z 769.87,A -85,B 0,C 180,E1 -28648.569,E2 -28648.569} C_VEL
LIN {X 0,Y 68.11,Z 768.258,A -85,B 0,C 180,E1 -28638.034,E2 -28638.034} C_VEL
LIN {X 0,Y 78.824,Z 765.511,A -85,B 0,C 180,E1 -28630.273,E2 -28630.273} C_VEL
LIN {X 0,Y 91.586,Z 761.151,A -85,B 0,C 180,E1 -28624.033,E2 -28624.033} C_VEL
LIN {X 0,Y 105.423,Z 755.089,A -85,B 0,C 180,E1 -28619.303,E2 -28619.303} C_VEL
LIN {X 0,Y 117.557,Z 748.579,A -85,B 0,C 180,E1 -28616.174,E2 -28616.174} C_VEL
LIN {X 0,Y 129.246,Z 741.136,A -85,B 0,C 180,E1 -28613.757,E2 -28613.757} C_VEL
LIN {X 0,Y 140.179,Z 732.951,A -85,B 0,C 180,E1 -28611.948,E2 -28611.948} C_VEL
LIN {X 0,Y 151.497,Z 722.952,A -85,B 0,C 180,E1 -28610.318,E2 -28610.318} C_VEL
LIN {X 0,Y 157.211,Z 717.228,A -85,B 0,C 180,E1 -28609.564,E2 -28609.564} C_VEL
LIN {X 0,Y 149.845,Z 724.584,A -85,B 0,C 180,E1 -28608.727,E2 -28608.727} C_VEL
LIN {X 0,Y 145.191,Z 728.832,A -85,B 0,C 180,E1 -28608.5,E2 -28608.5} C_VEL
LIN {X 0,Y 138.718,Z 734.162,A -85,B 0,C 180,E1 -28608.902,E2 -28608.902} C_VEL
LIN {X 0,Y 130.386,Z 740.252,A -85,B 0,C 180,E1 -28610.154,E2 -28610.154} C_VEL
LIN {X 0,Y 123.551,Z 744.769,A -85,B 0,C 180,E1 -28611.367,E2 -28611.367} C_VEL
LIN {X 0,Y 113.21,Z 750.821,A -85,B 0,C 180,E1 -28613.328,E2 -28613.328} C_VEL
LIN {X 0,Y 101.545,Z 756.618,A -85,B 0,C 180,E1 -28616.032,E2 -28616.032} C_VEL
LIN {X 0,Y 88.452,Z 761.895,A -85,B 0,C 180,E1 -28620.001,E2 -28620.001} C_VEL
LIN {X 0,Y 76.056,Z 765.811,A -85,B 0,C 180,E1 -28625.303,E2 -28625.303} C_VEL
LIN {X 0,Y 64.455,Z 768.533,A -85,B 0,C 180,E1 -28632.598,E2 -28632.598} C_VEL
LIN {X 0,Y 53.648,Z 770.146,A -85,B 0,C 180,E1 -28643.518,E2 -28643.518} C_VEL
LIN {X 0,Y 45.32,Z 770.452,A -85,B 0,C 180,E1 -28659.169,E2 -28659.169} C_VEL
LIN {X 0,Y 40.979,Z 769.434,A -85,B 0,C 180,E1 -28679.043,E2 -28679.043} C_VEL
LIN {X 0,Y 40.538,Z 768.444,A -85,B 0,C 180,E1 -28689.718,E2 -28689.718} C_VEL
LIN {X 0,Y 43.065,Z 765.505,A -85,B 0,C 180,E1 -28710.005,E2 -28710.005} C_VEL
LIN {X 0,Y 49.244,Z 761.272,A -85,B 0,C 180,E1 -28726.59,E2 -28726.59} C_VEL
LIN {X 0,Y 58.021,Z 755.653,A -85,B 0,C 180,E1 -28738.985,E2 -28738.985} C_VEL
LIN {X 0,Y 68.531,Z 748.485,A -85,B 0,C 180,E1 -28747.978,E2 -28747.978} C_VEL
LIN {X 0,Y 78.887,Z 740.593,A -85,B 0,C 180,E1 -28753.953,E2 -28753.953} C_VEL
LIN {X 0,Y 89.332,Z 731.502,A -85,B 0,C 180,E1 -28758.368,E2 -28758.368} C_VEL
LIN {X 0,Y 100.418,Z 720.26,A -85,B 0,C 180,E1 -28761.942,E2 -28761.942} C_VEL
LIN {X 0,Y 110.498,Z 708.22,A -85,B 0,C 180,E1 -28764.508,E2 -28764.508} C_VEL
LIN {X 0,Y 119.212,Z 695.902,A -85,B 0,C 180,E1 -28766.382,E2 -28766.382} C_VEL
LIN {X 0,Y 126.685,Z 683.368,A -85,B 0,C 180,E1 -28767.783,E2 -28767.783} C_VEL
LIN {X 0,Y 133.34,Z 669.822,A -85,B 0,C 180,E1 -28768.927,E2 -28768.927} C_VEL
LIN {X 0,Y 138.914,Z 655.648,A -85,B 0,C 180,E1 -28769.813,E2 -28769.813} C_VEL
LIN {X 0,Y 143.702,Z 639.575,A -85,B 0,C 180,E1 -28770.506,E2 -28770.506} C_VEL
LIN {X 0,Y 146.884,Z 624.197,A -85,B 0,C 180,E1 -28770.936,E2 -28770.936} C_VEL
LIN {X 0,Y 149.772,Z 601.492,A -85,B 0,C 180,E1 -28771.449,E2 -28771.449} C_VEL
LIN {X 0,Y 147.988,Z 596.217,A -85,B 0,C 180,E1 -28775.378,E2 -28775.378} C_VEL
LIN {X 0,Y 146.566,Z 592.089,A -85,B 0,C 180,E1 -28779.627,E2 -28779.627} C_VEL
LIN {X 0,Y 145.634,Z 589.149,A -85,B 0,C 180,E1 -28784.49,E2 -28784.49} C_VEL
LIN {X 0,Y 145.361,Z 588.577,A -85,B 0,C 180,E1 -28788.848,E2 -28788.848} C_VEL
LIN {X 0,Y 145.8,Z 589.075,A -85,B 0,C 180,E1 -28793.881,E2 -28793.881} C_VEL
LIN {X 0,Y 146.748,Z 592.289,A -85,B 0,C 180,E1 -28798.507,E2 -28798.507} C_VEL
LIN {X 0,Y 147.922,Z 595.669,A -85,B 0,C 180,E1 -28801.941,E2 -28801.941} C_VEL
LIN {X 0,Y 149.871,Z 601.671,A -85,B 0,C 180,E1 -28806.297,E2 -28806.297} C_VEL
LIN {X 0,Y 146.224,Z 629.209,A -85,B 0,C 180,E1 -28806.869,E2 -28806.869} C_VEL
LIN {X 0,Y 142.859,Z 644.459,A -85,B 0,C 180,E1 -28807.33,E2 -28807.33} C_VEL
LIN {X 0,Y 138.345,Z 658.844,A -85,B 0,C 180,E1 -28807.852,E2 -28807.852} C_VEL
LIN {X 0,Y 132.42,Z 673.489,A -85,B 0,C 180,E1 -28808.692,E2 -28808.692} C_VEL
LIN {X 0,Y 125.742,Z 686.712,A -85,B 0,C 180,E1 -28809.697,E2 -28809.697} C_VEL
LIN {X 0,Y 118.976,Z 697.889,A -85,B 0,C 180,E1 -28810.865,E2 -28810.865} C_VEL
LIN {X 0,Y 109.857,Z 710.693,A -85,B 0,C 180,E1 -28812.676,E2 -28812.676} C_VEL
LIN {X 0,Y 100.076,Z 722.32,A -85,B 0,C 180,E1 -28815.062,E2 -28815.062} C_VEL
LIN {X 0,Y 90.339,Z 732.23,A -85,B 0,C 180,E1 -28817.998,E2 -28817.998} C_VEL
LIN {X 0,Y 81.217,Z 740.39,A -85,B 0,C 180,E1 -28821.522,E2 -28821.522} C_VEL
LIN {X 0,Y 72.359,Z 747.518,A -85,B 0,C 180,E1 -28826.043,E2 -28826.043} C_VEL
LIN {X 0,Y 62.668,Z 754.406,A -85,B 0,C 180,E1 -28832.738,E2 -28832.738} C_VEL
LIN {X 0,Y 53.004,Z 760.764,A -85,B 0,C 180,E1 -28843.17,E2 -28843.17} C_VEL
LIN {X 0,Y 45.658,Z 765.646,A -85,B 0,C 180,E1 -28857.397,E2 -28857.397} C_VEL
LIN {X 0,Y 42.341,Z 768.449,A -85,B 0,C 180,E1 -28870.606,E2 -28870.606} C_VEL
LIN {X 0,Y 41.345,Z 769.902,A -85,B 0,C 180,E1 -28880.208,E2 -28880.208} C_VEL
LIN {X 0,Y 41.285,Z 771.018,A -85,B 0,C 180,E1 -28889.995,E2 -28889.995} C_VEL
LIN {X 0,Y 42.333,Z 772.268,A -85,B 0,C 180,E1 -28909.387,E2 -28909.387} C_VEL
LIN {X 0,Y 47.273,Z 772.434,A -85,B 0,C 180,E1 -28926.483,E2 -28926.483} C_VEL
LIN {X 0,Y 55.425,Z 771.554,A -85,B 0,C 180,E1 -28939.528,E2 -28939.528} C_VEL
LIN {X 0,Y 65.657,Z 769.568,A -85,B 0,C 180,E1 -28948.899,E2 -28948.899} C_VEL
LIN {X 0,Y 77.167,Z 766.465,A -85,B 0,C 180,E1 -28955.6,E2 -28955.6} C_VEL
LIN {X 0,Y 89.524,Z 762.211,A -85,B 0,C 180,E1 -28960.389,E2 -28960.389} C_VEL
LIN {X 0,Y 102.267,Z 756.738,A -85,B 0,C 180,E1 -28964.167,E2 -28964.167} C_VEL
LIN {X 0,Y 115.457,Z 749.859,A -85,B 0,C 180,E1 -28966.878,E2 -28966.878} C_VEL
LIN {X 0,Y 128.861,Z 741.39,A -85,B 0,C 180,E1 -28969.011,E2 -28969.011} C_VEL
LIN {X 0,Y 130.583,Z 740.161,A -85,B 0,C 180,E1 -28969.234,E2 -28969.234} C_VEL
LIN {X 0,Y 132.057,Z 739.079,A -85,B 0,C 180,E1 -28970.048,E2 -28970.048} C_VEL
LIN {X 0,Y 123.551,Z 744.769,A -85,B 0,C 180,E1 -28971.367,E2 -28971.367} C_VEL
LIN {X 0,Y 118.596,Z 747.795,A -85,B 0,C 180,E1 -28971.905,E2 -28971.905} C_VEL
LIN {X 0,Y 109.878,Z 752.534,A -85,B 0,C 180,E1 -28972.047,E2 -28972.047} C_VEL
LIN {X 0,Y 100.942,Z 756.803,A -85,B 0,C 180,E1 -28972.266,E2 -28972.266} C_VEL
LIN {X 0,Y 95.667,Z 758.989,A -85,B 0,C 180,E1 -28973.065,E2 -28973.065} C_VEL
LIN {X 0,Y 84.527,Z 763.039,A -85,B 0,C 180,E1 -28976.098,E2 -28976.098} C_VEL
LIN {X 0,Y 70.303,Z 767.007,A -85,B 0,C 180,E1 -28981.601,E2 -28981.601} C_VEL
LIN {X 0,Y 57.038,Z 769.527,A -85,B 0,C 180,E1 -28989.72,E2 -28989.72} C_VEL
LIN {X 0,Y 45.485,Z 770.662,A -85,B 0,C 180,E1 -29002.032,E2 -29002.032} C_VEL
LIN {X 0,Y 37.028,Z 770.449,A -85,B 0,C 180,E1 -29020.616,E2 -29020.616} C_VEL
LIN {X 0,Y 33.452,Z 768.931,A -85,B 0,C 180,E1 -29045.161,E2 -29045.161} C_VEL
LIN {X 0,Y 35.597,Z 766.126,A -85,B 0,C 180,E1 -29070.006,E2 -29070.006} C_VEL
LIN {X 0,Y 42.253,Z 762.018,A -85,B 0,C 180,E1 -29089.436,E2 -29089.436} C_VEL
LIN {X 0,Y 51.775,Z 756.548,A -85,B 0,C 180,E1 -29102.89,E2 -29102.89} C_VEL
LIN {X 0,Y 62.977,Z 749.572,A -85,B 0,C 180,E1 -29112.039,E2 -29112.039} C_VEL
LIN {X 0,Y 73.466,Z 742.109,A -85,B 0,C 180,E1 -29117.712,E2 -29117.712} C_VEL
LIN {X 0,Y 84.703,Z 732.942,A -85,B 0,C 180,E1 -29122.025,E2 -29122.025} C_VEL
LIN {X 0,Y 94.464,Z 723.68,A -85,B 0,C 180,E1 -29124.927,E2 -29124.927} C_VEL
LIN {X 0,Y 104.372,Z 712.791,A -85,B 0,C 180,E1 -29127.251,E2 -29127.251} C_VEL
LIN {X 0,Y 113.682,Z 700.726,A -85,B 0,C 180,E1 -29129.07,E2 -29129.07} C_VEL
LIN {X 0,Y 122.152,Z 687.627,A -85,B 0,C 180,E1 -29130.486,E2 -29130.486} C_VEL
LIN {X 0,Y 128.919,Z 674.989,A -85,B 0,C 180,E1 -29131.53,E2 -29131.53} C_VEL
LIN {X 0,Y 134.875,Z 661.389,A -85,B 0,C 180,E1 -29132.355,E2 -29132.355} C_VEL
LIN {X 0,Y 139.898,Z 646.697,A -85,B 0,C 180,E1 -29133.018,E2 -29133.018} C_VEL
LIN {X 0,Y 143.676,Z 631.666,A -85,B 0,C 180,E1 -29133.479,E2 -29133.479} C_VEL
LIN {X 0,Y 146.36,Z 615.062,A -85,B 0,C 180,E1 -29133.803,E2 -29133.803} C_VEL
LIN {X 0,Y 147.491,Z 605.62,A -85,B 0,C 180,E1 -29134.044,E2 -29134.044} C_VEL
LIN {X 0,Y 146.086,Z 601.069,A -85,B 0,C 180,E1 -29137.855,E2 -29137.855} C_VEL
LIN {X 0,Y 145.285,Z 598.607,A -85,B 0,C 180,E1 -29140.866,E2 -29140.866} C_VEL
LIN {X 0,Y 144.654,Z 596.144,A -85,B 0,C 180,E1 -29144.827,E2 -29144.827} C_VEL
LIN {X 0,Y 144.435,Z 595.611,A -85,B 0,C 180,E1 -29148.776,E2 -29148.776} C_VEL
LIN {X 0,Y 144.762,Z 595.981,A -85,B 0,C 180,E1 -29153.247,E2 -29153.247} C_VEL
LIN {X 0,Y 145.499,Z 598.761,A -85,B 0,C 180,E1 -29157.452,E2 -29157.452} C_VEL
LIN {X 0,Y 146.653,Z 602.576,A -85,B 0,C 180,E1 -29161.311,E2 -29161.311} C_VEL
LIN {X 0,Y 147.557,Z 605.994,A -85,B 0,C 180,E1 -29163.738,E2 -29163.738} C_VEL
LIN {X 0,Y 144.251,Z 629.842,A -85,B 0,C 180,E1 -29164.193,E2 -29164.193} C_VEL
LIN {X 0,Y 140.794,Z 644.944,A -85,B 0,C 180,E1 -29164.59,E2 -29164.59} C_VEL
LIN {X 0,Y 136.256,Z 659.086,A -85,B 0,C 180,E1 -29165.034,E2 -29165.034} C_VEL
LIN {X 0,Y 130.665,Z 672.738,A -85,B 0,C 180,E1 -29165.696,E2 -29165.696} C_VEL
LIN {X 0,Y 123.787,Z 686.203,A -85,B 0,C 180,E1 -29166.565,E2 -29166.565} C_VEL
LIN {X 0,Y 116.982,Z 697.288,A -85,B 0,C 180,E1 -29167.564,E2 -29167.564} C_VEL
LIN {X 0,Y 107.662,Z 710.156,A -85,B 0,C 180,E1 -29169.12,E2 -29169.12} C_VEL
LIN {X 0,Y 98.453,Z 720.933,A -85,B 0,C 180,E1 -29171.019,E2 -29171.019} C_VEL
LIN {X 0,Y 88.542,Z 730.883,A -85,B 0,C 180,E1 -29173.499,E2 -29173.499} C_VEL
LIN {X 0,Y 78.856,Z 739.363,A -85,B 0,C 180,E1 -29176.64,E2 -29176.64} C_VEL
LIN {X 0,Y 67.968,Z 747.683,A -85,B 0,C 180,E1 -29181.462,E2 -29181.462} C_VEL
LIN {X 0,Y 56.263,Z 755.393,A -85,B 0,C 180,E1 -29189.02,E2 -29189.02} C_VEL
LIN {X 0,Y 45.976,Z 761.496,A -85,B 0,C 180,E1 -29200.148,E2 -29200.148} C_VEL
LIN {X 0,Y 38.155,Z 766.159,A -85,B 0,C 180,E1 -29216.449,E2 -29216.449} C_VEL
LIN {X 0,Y 34.341,Z 769.462,A -85,B 0,C 180,E1 -29238.184,E2 -29238.184} C_VEL
LIN {X 0,Y 34.185,Z 770.627,A -85,B 0,C 180,E1 -29249.993,E2 -29249.993} C_VEL
LIN {X 0,Y 35.677,Z 771.979,A -85,B 0,C 180,E1 -29273.196,E2 -29273.196} C_VEL
LIN {X 0,Y 41.746,Z 772.253,A -85,B 0,C 180,E1 -29292.323,E2 -29292.323} C_VEL
LIN {X 0,Y 51.066,Z 771.466,A -85,B 0,C 180,E1 -29305.657,E2 -29305.657} C_VEL
LIN {X 0,Y 62.263,Z 769.556,A -85,B 0,C 180,E1 -29314.546,E2 -29314.546} C_VEL
LIN {X 0,Y 74.497,Z 766.58,A -85,B 0,C 180,E1 -29320.619,E2 -29320.619} C_VEL
LIN {X 0,Y 87.39,Z 762.467,A -85,B 0,C 180,E1 -29324.795,E2 -29324.795} C_VEL
LIN {X 0,Y 100.563,Z 757.131,A -85,B 0,C 180,E1 -29328.06,E2 -29328.06} C_VEL
LIN {X 0,Y 107.291,Z 753.94,A -85,B 0,C 180,E1 -29329.27,E2 -29329.27} C_VEL
LIN {X 0,Y 109.479,Z 752.77,A -85,B 0,C 180,E1 -29330.201,E2 -29330.201} C_VEL
LIN {X 0,Y 95.667,Z 758.989,A -85,B 0,C 180,E1 -29333.065,E2 -29333.065} C_VEL
LIN {X 0,Y 90.328,Z 761.047,A -85,B 0,C 180,E1 -29333.971,E2 -29333.971} C_VEL
LIN {X 0,Y 80.942,Z 764.125,A -85,B 0,C 180,E1 -29334.549,E2 -29334.549} C_VEL
LIN {X 0,Y 73.315,Z 766.212,A -85,B 0,C 180,E1 -29335.057,E2 -29335.057} C_VEL
LIN {X 0,Y 67.729,Z 767.501,A -85,B 0,C 180,E1 -29336.186,E2 -29336.186} C_VEL
LIN {X 0,Y 65.951,Z 767.863,A -85,B 0,C 180,E1 -29336.826,E2 -29336.826} C_VEL
LIN {X 0,Y 56.242,Z 769.574,A -85,B 0,C 180,E1 -29341.615,E2 -29341.615} C_VEL
LIN {X 0,Y 43.137,Z 770.843,A -85,B 0,C 180,E1 -29352.194,E2 -29352.194} C_VEL
LIN {X 0,Y 32.449,Z 770.757,A -85,B 0,C 180,E1 -29369.979,E2 -29369.979} C_VEL
LIN {X 0,Y 26.661,Z 769.354,A -85,B 0,C 180,E1 -29398.193,E2 -29398.193} C_VEL
LIN {X 0,Y 28.114,Z 766.65,A -85,B 0,C 180,E1 -29430.191,E2 -29430.191} C_VEL
LIN {X 0,Y 35.377,Z 762.705,A -85,B 0,C 180,E1 -29453.417,E2 -29453.417} C_VEL
LIN {X 0,Y 45.836,Z 757.384,A -85,B 0,C 180,E1 -29467.835,E2 -29467.835} C_VEL
LIN {X 0,Y 57.772,Z 750.579,A -85,B 0,C 180,E1 -29476.883,E2 -29476.883} C_VEL
LIN {X 0,Y 68.651,Z 743.408,A -85,B 0,C 180,E1 -29482.102,E2 -29482.102} C_VEL
LIN {X 0,Y 80.458,Z 734.334,A -85,B 0,C 180,E1 -29486.085,E2 -29486.085} C_VEL
LIN {X 0,Y 92.198,Z 723.642,A -85,B 0,C 180,E1 -29489.047,E2 -29489.047} C_VEL
LIN {X 0,Y 102.886,Z 712.092,A -85,B 0,C 180,E1 -29491.108,E2 -29491.108} C_VEL
LIN {X 0,Y 111.857,Z 700.59,A -85,B 0,C 180,E1 -29492.56,E2 -29492.56} C_VEL
LIN {X 0,Y 120.482,Z 687.419,A -85,B 0,C 180,E1 -29493.751,E2 -29493.751} C_VEL
LIN {X 0,Y 127.366,Z 674.682,A -85,B 0,C 180,E1 -29494.633,E2 -29494.633} C_VEL
LIN {X 0,Y 133.63,Z 660.374,A -85,B 0,C 180,E1 -29495.353,E2 -29495.353} C_VEL
LIN {X 0,Y 138.794,Z 645.02,A -85,B 0,C 180,E1 -29495.932,E2 -29495.932} C_VEL
LIN {X 0,Y 142.619,Z 629.171,A -85,B 0,C 180,E1 -29496.302,E2 -29496.302} C_VEL
LIN {X 0,Y 145.453,Z 610.054,A -85,B 0,C 180,E1 -29496.644,E2 -29496.644} C_VEL
LIN {X 0,Y 144.569,Z 606.849,A -85,B 0,C 180,E1 -29499.719,E2 -29499.719} C_VEL
LIN {X 0,Y 144.054,Z 605.044,A -85,B 0,C 180,E1 -29502.17,E2 -29502.17} C_VEL
LIN {X 0,Y 143.665,Z 603.121,A -85,B 0,C 180,E1 -29505.282,E2 -29505.282} C_VEL
LIN {X 0,Y 143.507,Z 602.659,A -85,B 0,C 180,E1 -29508.702,E2 -29508.702} C_VEL
LIN {X 0,Y 143.782,Z 602.992,A -85,B 0,C 180,E1 -29512.944,E2 -29512.944} C_VEL
LIN {X 0,Y 144.422,Z 605.829,A -85,B 0,C 180,E1 -29517.038,E2 -29517.038} C_VEL
LIN {X 0,Y 145.267,Z 609.021,A -85,B 0,C 180,E1 -29520.259,E2 -29520.259} C_VEL
LIN {X 0,Y 145.523,Z 610.109,A -85,B 0,C 180,E1 -29521.083,E2 -29521.083} C_VEL
LIN {X 0,Y 142.465,Z 630.979,A -85,B 0,C 180,E1 -29521.461,E2 -29521.461} C_VEL
LIN {X 0,Y 138.654,Z 646.694,A -85,B 0,C 180,E1 -29521.797,E2 -29521.797} C_VEL
LIN {X 0,Y 133.634,Z 661.496,A -85,B 0,C 180,E1 -29522.214,E2 -29522.214} C_VEL
LIN {X 0,Y 127.539,Z 675.49,A -85,B 0,C 180,E1 -29522.819,E2 -29522.819} C_VEL
LIN {X 0,Y 120.483,Z 688.514,A -85,B 0,C 180,E1 -29523.51,E2 -29523.51} C_VEL
LIN {X 0,Y 114.52,Z 697.923,A -85,B 0,C 180,E1 -29524.236,E2 -29524.236} C_VEL
LIN {X 0,Y 105.039,Z 710.662,A -85,B 0,C 180,E1 -29525.563,E2 -29525.563} C_VEL
LIN {X 0,Y 95.628,Z 721.322,A -85,B 0,C 180,E1 -29527.168,E2 -29527.168} C_VEL
LIN {X 0,Y 85.46,Z 731.176,A -85,B 0,C 180,E1 -29529.292,E2 -29529.292} C_VEL
LIN {X 0,Y 75.447,Z 739.57,A -85,B 0,C 180,E1 -29532.005,E2 -29532.005} C_VEL
LIN {X 0,Y 64.077,Z 747.819,A -85,B 0,C 180,E1 -29536.311,E2 -29536.311} C_VEL
LIN {X 0,Y 53.146,Z 754.615,A -85,B 0,C 180,E1 -29542.221,E2 -29542.221} C_VEL
LIN {X 0,Y 41.71,Z 760.84,A -85,B 0,C 180,E1 -29552.588,E2 -29552.588} C_VEL
LIN {X 0,Y 32.431,Z 765.595,A -85,B 0,C 180,E1 -29569.441,E2 -29569.441} C_VEL
LIN {X 0,Y 27.39,Z 769.006,A -85,B 0,C 180,E1 -29595.124,E2 -29595.124} C_VEL
LIN {X 0,Y 27.069,Z 770.227,A -85,B 0,C 180,E1 -29609.992,E2 -29609.992} C_VEL
LIN {X 0,Y 29.256,Z 771.687,A -85,B 0,C 180,E1 -29638.706,E2 -29638.706} C_VEL
LIN {X 0,Y 36.762,Z 772.071,A -85,B 0,C 180,E1 -29659.87,E2 -29659.87} C_VEL
LIN {X 0,Y 47.387,Z 771.342,A -85,B 0,C 180,E1 -29672.844,E2 -29672.844} C_VEL
LIN {X 0,Y 59.537,Z 769.556,A -85,B 0,C 180,E1 -29680.781,E2 -29680.781} C_VEL
LIN {X 0,Y 72.438,Z 766.706,A -85,B 0,C 180,E1 -29685.963,E2 -29685.963} C_VEL
LIN {X 0,Y 85.796,Z 762.723,A -85,B 0,C 180,E1 -29689.396,E2 -29689.396} C_VEL
LIN {X 0,Y 86.005,Z 762.605,A -85,B 0,C 180,E1 -29690.595,E2 -29690.595} C_VEL
LIN {X 0,Y 72.345,Z 766.464,A -85,B 0,C 180,E1 -29694.427,E2 -29694.427} C_VEL
LIN {X 0,Y 65.951,Z 767.863,A -85,B 0,C 180,E1 -29696.826,E2 -29696.826} C_VEL
LIN {X 0,Y 60.473,Z 768.902,A -85,B 0,C 180,E1 -29698.614,E2 -29698.614} C_VEL
LIN {X 0,Y 50.816,Z 770.226,A -85,B 0,C 180,E1 -29700.542,E2 -29700.542} C_VEL
LIN {X 0,Y 43.049,Z 770.896,A -85,B 0,C 180,E1 -29702.522,E2 -29702.522} C_VEL
LIN {X 0,Y 37.548,Z 771.128,A -85,B 0,C 180,E1 -29705.634,E2 -29705.634} C_VEL
LIN {X 0,Y 35.866,Z 771.152,A -85,B 0,C 180,E1 -29707.247,E2 -29707.247} C_VEL
LIN {X 0,Y 24.109,Z 770.555,A -85,B 0,C 180,E1 -29729.029,E2 -29729.029} C_VEL
LIN {X 0,Y 20.522,Z 769.76,A -85,B 0,C 180,E1 -29746.787,E2 -29746.787} C_VEL
LIN {X 0,Y 20.512,Z 767.217,A -85,B 0,C 180,E1 -29790.011,E2 -29790.011} C_VEL
LIN {X 0,Y 26.238,Z 764.506,A -85,B 0,C 180,E1 -29813.698,E2 -29813.698} C_VEL
LIN {X 0,Y 37.67,Z 759.493,A -85,B 0,C 180,E1 -29831.727,E2 -29831.727} C_VEL
LIN {X 0,Y 49.804,Z 753.42,A -85,B 0,C 180,E1 -29840.913,E2 -29840.913} C_VEL
LIN {X 0,Y 63.052,Z 745.531,A -85,B 0,C 180,E1 -29846.728,E2 -29846.728} C_VEL
LIN {X 0,Y 74.935,Z 737.081,A -85,B 0,C 180,E1 -29850.179,E2 -29850.179} C_VEL
LIN {X 0,Y 86.966,Z 726.907,A -85,B 0,C 180,E1 -29852.745,E2 -29852.745} C_VEL
LIN {X 0,Y 98.118,Z 715.658,A -85,B 0,C 180,E1 -29854.546,E2 -29854.546} C_VEL
LIN {X 0,Y 107.841,Z 703.991,A -85,B 0,C 180,E1 -29855.84,E2 -29855.84} C_VEL
LIN {X 0,Y 116.584,Z 691.48,A -85,B 0,C 180,E1 -29856.829,E2 -29856.829} C_VEL
LIN {X 0,Y 124.453,Z 677.848,A -85,B 0,C 180,E1 -29857.629,E2 -29857.629} C_VEL
LIN {X 0,Y 131.239,Z 663.228,A -85,B 0,C 180,E1 -29858.248,E2 -29858.248} C_VEL
LIN {X 0,Y 136.819,Z 647.555,A -85,B 0,C 180,E1 -29858.755,E2 -29858.755} C_VEL
LIN {X 0,Y 140.76,Z 632.395,A -85,B 0,C 180,E1 -29859.072,E2 -29859.072} C_VEL
LIN {X 0,Y 143.534,Z 615.8,A -85,B 0,C 180,E1 -29859.289,E2 -29859.289} C_VEL
LIN {X 0,Y 143.655,Z 614.569,A -85,B 0,C 180,E1 -29859.406,E2 -29859.406} C_VEL
LIN {X 0,Y 143.01,Z 611.965,A -85,B 0,C 180,E1 -29862.647,E2 -29862.647} C_VEL
LIN {X 0,Y 142.687,Z 610.089,A -85,B 0,C 180,E1 -29865.742,E2 -29865.742} C_VEL
LIN {X 0,Y 142.602,Z 609.735,A -85,B 0,C 180,E1 -29870.298,E2 -29870.298} C_VEL
LIN {X 0,Y 142.827,Z 610.233,A -85,B 0,C 180,E1 -29872.955,E2 -29872.955} C_VEL
LIN {X 0,Y 143.306,Z 612.603,A -85,B 0,C 180,E1 -29876.323,E2 -29876.323} C_VEL
LIN {X 0,Y 143.733,Z 614.491,A -85,B 0,C 180,E1 -29878.362,E2 -29878.362} C_VEL
LIN {X 0,Y 141.072,Z 631.558,A -85,B 0,C 180,E1 -29878.648,E2 -29878.648} C_VEL
LIN {X 0,Y 137.225,Z 647.034,A -85,B 0,C 180,E1 -29878.92,E2 -29878.92} C_VEL
LIN {X 0,Y 132.229,Z 661.525,A -85,B 0,C 180,E1 -29879.225,E2 -29879.225} C_VEL
LIN {X 0,Y 126.509,Z 674.576,A -85,B 0,C 180,E1 -29879.654,E2 -29879.654} C_VEL
LIN {X 0,Y 119.479,Z 687.573,A -85,B 0,C 180,E1 -29880.156,E2 -29880.156} C_VEL
LIN {X 0,Y 113.338,Z 697.206,A -85,B 0,C 180,E1 -29880.733,E2 -29880.733} C_VEL
LIN {X 0,Y 103.714,Z 710.029,A -85,B 0,C 180,E1 -29881.745,E2 -29881.745} C_VEL
LIN {X 0,Y 93.261,Z 721.664,A -85,B 0,C 180,E1 -29883.105,E2 -29883.105} C_VEL
LIN {X 0,Y 82.323,Z 731.911,A -85,B 0,C 180,E1 -29884.896,E2 -29884.896} C_VEL
LIN {X 0,Y 70.883,Z 741.011,A -85,B 0,C 180,E1 -29887.459,E2 -29887.459} C_VEL
LIN {X 0,Y 59.095,Z 748.95,A -85,B 0,C 180,E1 -29891.127,E2 -29891.127} C_VEL
LIN {X 0,Y 47.637,Z 755.499,A -85,B 0,C 180,E1 -29896.474,E2 -29896.474} C_VEL
LIN {X 0,Y 35.392,Z 761.483,A -85,B 0,C 180,E1 -29906.66,E2 -29906.66} C_VEL
LIN {X 0,Y 27.394,Z 765.01,A -85,B 0,C 180,E1 -29919.664,E2 -29919.664} C_VEL
LIN {X 0,Y 20.582,Z 768.542,A -85,B 0,C 180,E1 -29950.022,E2 -29950.022} C_VEL
LIN {X 0,Y 19.964,Z 769.823,A -85,B 0,C 180,E1 -29969.989,E2 -29969.989} C_VEL
LIN {X 0,Y 23.231,Z 771.393,A -85,B 0,C 180,E1 -30007.221,E2 -30007.221} C_VEL
LIN {X 0,Y 32.608,Z 771.857,A -85,B 0,C 180,E1 -30029.54,E2 -30029.54} C_VEL
LIN {X 0,Y 47.066,Z 771.013,A -85,B 0,C 180,E1 -30042.626,E2 -30042.626} C_VEL
LIN {X 0,Y 64.275,Z 768.33,A -85,B 0,C 180,E1 -30049.74,E2 -30049.74} C_VEL
LIN {X 0,Y 64.079,Z 768.341,A -85,B 0,C 180,E1 -30050.761,E2 -30050.761} C_VEL
LIN {X 0,Y 49.263,Z 770.439,A -85,B 0,C 180,E1 -30056.91,E2 -30056.91} C_VEL
LIN {X 0,Y 35.866,Z 771.152,A -85,B 0,C 180,E1 -30067.247,E2 -30067.247} C_VEL
LIN {X 0,Y 30.771,Z 771.176,A -85,B 0,C 180,E1 -30072.4,E2 -30072.4} C_VEL
LIN {X 0,Y 21.865,Z 770.712,A -85,B 0,C 180,E1 -30082.007,E2 -30082.007} C_VEL
LIN {X 0,Y 15.354,Z 769.892,A -85,B 0,C 180,E1 -30096.426,E2 -30096.426} C_VEL
LIN {X 0,Y 12.322,Z 769.036,A -85,B 0,C 180,E1 -30117.68,E2 -30117.68} C_VEL
LIN {X 0,Y 12.034,Z 768.673,A -85,B 0,C 180,E1 -30126.82,E2 -30126.82} C_VEL
LIN {X 0,Y 16.969,Z 766.065,A -85,B 0,C 180,E1 -30174.482,E2 -30174.482} C_VEL
LIN {X 0,Y 28.862,Z 761.717,A -85,B 0,C 180,E1 -30196.941,E2 -30196.941} C_VEL
LIN {X 0,Y 38.782,Z 757.553,A -85,B 0,C 180,E1 -30204.645,E2 -30204.645} C_VEL
LIN {X 0,Y 52.443,Z 750.68,A -85,B 0,C 180,E1 -30210.593,E2 -30210.593} C_VEL
LIN {X 0,Y 64.032,Z 743.619,A -85,B 0,C 180,E1 -30213.723,E2 -30213.723} C_VEL
LIN {X 0,Y 76.871,Z 734.286,A -85,B 0,C 180,E1 -30216.106,E2 -30216.106} C_VEL
LIN {X 0,Y 87.406,Z 725.174,A -85,B 0,C 180,E1 -30217.624,E2 -30217.624} C_VEL
LIN {X 0,Y 98.014,Z 714.376,A -85,B 0,C 180,E1 -30218.778,E2 -30218.778} C_VEL
LIN {X 0,Y 107.751,Z 702.595,A -85,B 0,C 180,E1 -30219.656,E2 -30219.656} C_VEL
LIN {X 0,Y 116.601,Z 689.763,A -85,B 0,C 180,E1 -30220.356,E2 -30220.356} C_VEL
LIN {X 0,Y 124.541,Z 675.695,A -85,B 0,C 180,E1 -30220.952,E2 -30220.952} C_VEL
LIN {X 0,Y 130.994,Z 661.429,A -85,B 0,C 180,E1 -30221.376,E2 -30221.376} C_VEL
LIN {X 0,Y 136.205,Z 646.531,A -85,B 0,C 180,E1 -30221.722,E2 -30221.722} C_VEL
LIN {X 0,Y 139.897,Z 632.207,A -85,B 0,C 180,E1 -30221.948,E2 -30221.948} C_VEL
LIN {X 0,Y 142.11,Z 619.587,A -85,B 0,C 180,E1 -30222.121,E2 -30222.121} C_VEL
LIN {X 0,Y 141.699,Z 617.036,A -85,B 0,C 180,E1 -30226.457,E2 -30226.457} C_VEL
LIN {X 0,Y 141.654,Z 616.738,A -85,B 0,C 180,E1 -30228.553,E2 -30228.553} C_VEL
LIN {X 0,Y 141.826,Z 617.098,A -85,B 0,C 180,E1 -30232.344,E2 -30232.344} C_VEL
LIN {X 0,Y 142.197,Z 619.372,A -85,B 0,C 180,E1 -30235.555,E2 -30235.555} C_VEL
LIN {X 0,Y 139.595,Z 634.28,A -85,B 0,C 180,E1 -30235.809,E2 -30235.809} C_VEL
LIN {X 0,Y 135.545,Z 649.426,A -85,B 0,C 180,E1 -30236.012,E2 -30236.012} C_VEL
LIN {X 0,Y 129.862,Z 664.887,A -85,B 0,C 180,E1 -30236.231,E2 -30236.231} C_VEL
LIN {X 0,Y 123.206,Z 678.991,A -85,B 0,C 180,E1 -30236.598,E2 -30236.598} C_VEL
LIN {X 0,Y 116.13,Z 691.134,A -85,B 0,C 180,E1 -30236.939,E2 -30236.939} C_VEL
LIN {X 0,Y 107.282,Z 703.832,A -85,B 0,C 180,E1 -30237.494,E2 -30237.494} C_VEL
LIN {X 0,Y 98.445,Z 714.506,A -85,B 0,C 180,E1 -30238.164,E2 -30238.164} C_VEL
LIN {X 0,Y 87.862,Z 725.378,A -85,B 0,C 180,E1 -30239.183,E2 -30239.183} C_VEL
LIN {X 0,Y 75.56,Z 735.949,A -85,B 0,C 180,E1 -30240.707,E2 -30240.707} C_VEL
LIN {X 0,Y 63.342,Z 744.742,A -85,B 0,C 180,E1 -30243.002,E2 -30243.002} C_VEL
LIN {X 0,Y 49.532,Z 752.916,A -85,B 0,C 180,E1 -30246.641,E2 -30246.641} C_VEL
LIN {X 0,Y 36.067,Z 759.412,A -85,B 0,C 180,E1 -30252.995,E2 -30252.995} C_VEL
LIN {X 0,Y 23.479,Z 764.422,A -85,B 0,C 180,E1 -30266.086,E2 -30266.086} C_VEL
LIN {X 0,Y 14.101,Z 768.076,A -85,B 0,C 180,E1 -30300.089,E2 -30300.089} C_VEL
LIN {X 0,Y 12.85,Z 769.415,A -85,B 0,C 180,E1 -30329.983,E2 -30329.983} C_VEL
LIN {X 0,Y 14.111,Z 770.395,A -85,B 0,C 180,E1 -30359.853,E2 -30359.853} C_VEL
LIN {X 0,Y 23.481,Z 771.488,A -85,B 0,C 180,E1 -30393.865,E2 -30393.865} C_VEL
LIN {X 0,Y 36.112,Z 771.489,A -85,B 0,C 180,E1 -30406.649,E2 -30406.649} C_VEL
LIN {X 0,Y 42.791,Z 771.104,A -85,B 0,C 180,E1 -30410.176,E2 -30410.176} C_VEL
LIN {X 0,Y 42.999,Z 771.08,A -85,B 0,C 180,E1 -30410.595,E2 -30410.595} C_VEL
LIN {X 0,Y 28.111,Z 771.29,A -85,B 0,C 180,E1 -30420.828,E2 -30420.828} C_VEL
LIN {X 0,Y 15.77,Z 770.162,A -85,B 0,C 180,E1 -30446.995,E2 -30446.995} C_VEL
LIN {X 0,Y 12.034,Z 768.673,A -85,B 0,C 180,E1 -30486.82,E2 -30486.82} C_VEL
LIN {X 0,Y 12.195,Z 768.011,A -85,B 0,C 180,E1 -30505.158,E2 -30505.158} C_VEL
LIN {X 0,Y 14.493,Z 766.358,A -85,B 0,C 180,E1 -30537.412,E2 -30537.412} C_VEL
LIN {X 0,Y 22.24,Z 763.265,A -85,B 0,C 180,E1 -30565.234,E2 -30565.234} C_VEL
LIN {X 0,Y 27.337,Z 761.389,A -85,B 0,C 180,E1 -30571.085,E2 -30571.085} C_VEL
LIN {X 0,Y 29.148,Z 760.712,A -85,B 0,C 180,E1 -30572.123,E2 -30572.123} C_VEL
LIN {X 0,Y 42.166,Z 755.185,A -85,B 0,C 180,E1 -30576.46,E2 -30576.46} C_VEL
LIN {X 0,Y 56.401,Z 747.649,A -85,B 0,C 180,E1 -30579.165,E2 -30579.165} C_VEL
LIN {X 0,Y 68.876,Z 739.551,A -85,B 0,C 180,E1 -30580.717,E2 -30580.717} C_VEL
LIN {X 0,Y 81.356,Z 729.804,A -85,B 0,C 180,E1 -30581.857,E2 -30581.857} C_VEL
LIN {X 0,Y 93.064,Z 718.816,A -85,B 0,C 180,E1 -30582.633,E2 -30582.633} C_VEL
LIN {X 0,Y 103.658,Z 706.872,A -85,B 0,C 180,E1 -30583.275,E2 -30583.275} C_VEL
LIN {X 0,Y 112.583,Z 694.842,A -85,B 0,C 180,E1 -30583.701,E2 -30583.701} C_VEL
LIN {X 0,Y 120.602,Z 681.853,A -85,B 0,C 180,E1 -30584.059,E2 -30584.059} C_VEL
LIN {X 0,Y 127.716,Z 667.667,A -85,B 0,C 180,E1 -30584.369,E2 -30584.369} C_VEL
LIN {X 0,Y 133.306,Z 653.561,A -85,B 0,C 180,E1 -30584.612,E2 -30584.612} C_VEL
LIN {X 0,Y 137.923,Z 638.047,A -85,B 0,C 180,E1 -30584.797,E2 -30584.797} C_VEL
LIN {X 0,Y 140.671,Z 625.023,A -85,B 0,C 180,E1 -30584.952,E2 -30584.952} C_VEL
LIN {X 0,Y 140.613,Z 623.971,A -85,B 0,C 180,E1 -30587.171,E2 -30587.171} C_VEL
LIN {X 0,Y 140.705,Z 623.871,A -85,B 0,C 180,E1 -30591.381,E2 -30591.381} C_VEL
LIN {X 0,Y 140.765,Z 624.654,A -85,B 0,C 180,E1 -30592.782,E2 -30592.782} C_VEL
LIN {X 0,Y 137.537,Z 639.969,A -85,B 0,C 180,E1 -30592.956,E2 -30592.956} C_VEL
LIN {X 0,Y 133.204,Z 654.211,A -85,B 0,C 180,E1 -30593.018,E2 -30593.018} C_VEL
LIN {X 0,Y 127.418,Z 668.69,A -85,B 0,C 180,E1 -30593.142,E2 -30593.142} C_VEL
LIN {X 0,Y 121.009,Z 681.486,A -85,B 0,C 180,E1 -30593.329,E2 -30593.329} C_VEL
LIN {X 0,Y 114.011,Z 693.11,A -85,B 0,C 180,E1 -30593.53,E2 -30593.53} C_VEL
LIN {X 0,Y 106.055,Z 704.236,A -85,B 0,C 180,E1 -30593.74,E2 -30593.74} C_VEL
LIN {X 0,Y 95.373,Z 716.798,A -85,B 0,C 180,E1 -30594.173,E2 -30594.173} C_VEL
LIN {X 0,Y 84.699,Z 727.257,A -85,B 0,C 180,E1 -30594.716,E2 -30594.716} C_VEL
LIN {X 0,Y 74.035,Z 736.098,A -85,B 0,C 180,E1 -30595.4,E2 -30595.4} C_VEL
LIN {X 0,Y 61.602,Z 744.825,A -85,B 0,C 180,E1 -30596.672,E2 -30596.672} C_VEL
LIN {X 0,Y 49.22,Z 752.025,A -85,B 0,C 180,E1 -30598.321,E2 -30598.321} C_VEL
LIN {X 0,Y 35.156,Z 758.666,A -85,B 0,C 180,E1 -30601.53,E2 -30601.53} C_VEL
LIN {X 0,Y 21.323,Z 763.811,A -85,B 0,C 180,E1 -30608.526,E2 -30608.526} C_VEL
LIN {X 0,Y 8.673,Z 767.594,A -85,B 0,C 180,E1 -30635.828,E2 -30635.828} C_VEL
LIN {X 0,Y 5.729,Z 768.996,A -85,B 0,C 180,E1 -30689.961,E2 -30689.961} C_VEL
LIN {X 0,Y 8.695,Z 770.029,A -85,B 0,C 180,E1 -30743.888,E2 -30743.888} C_VEL
LIN {X 0,Y 14.664,Z 770.743,A -85,B 0,C 180,E1 -30763.389,E2 -30763.389} C_VEL
LIN {X 0,Y 17.979,Z 770.955,A -85,B 0,C 180,E1 -30772.21,E2 -30772.21} C_VEL
LIN {X 0,Y 7.445,Z 769.584,A -85,B 0,C 180,E1 -30799.363,E2 -30799.363} C_VEL
LIN {X 0,Y 10.618,Z 766.659,A -85,B 0,C 180,E1 -30911.472,E2 -30911.472} C_VEL
LIN {X 0,Y 24.431,Z 762.444,A -85,B 0,C 180,E1 -30929.673,E2 -30929.673} C_VEL
LIN {X 0,Y 29.148,Z 760.712,A -85,B 0,C 180,E1 -30932.123,E2 -30932.123} C_VEL
LIN {X 0,Y 34.383,Z 758.628,A -85,B 0,C 180,E1 -30935.311,E2 -30935.311} C_VEL
LIN {X 0,Y 42.608,Z 754.822,A -85,B 0,C 180,E1 -30941.336,E2 -30941.336} C_VEL
LIN {X 0,Y 50.914,Z 750.564,A -85,B 0,C 180,E1 -30945.523,E2 -30945.523} C_VEL
LIN {X 0,Y 56.04,Z 747.642,A -85,B 0,C 180,E1 -30946.39,E2 -30946.39} C_VEL
LIN {X 0,Y 68.631,Z 739.493,A -85,B 0,C 180,E1 -30946.623,E2 -30946.623} C_VEL
LIN {X 0,Y 79.408,Z 731.209,A -85,B 0,C 180,E1 -30946.802,E2 -30946.802} C_VEL
LIN {X 0,Y 90.174,Z 721.476,A -85,B 0,C 180,E1 -30946.971,E2 -30946.971} C_VEL
LIN {X 0,Y 100.93,Z 709.883,A -85,B 0,C 180,E1 -30947.13,E2 -30947.13} C_VEL
LIN {X 0,Y 110.776,Z 697.124,A -85,B 0,C 180,E1 -30947.281,E2 -30947.281} C_VEL
LIN {X 0,Y 118.827,Z 684.589,A -85,B 0,C 180,E1 -30947.398,E2 -30947.398} C_VEL
LIN {X 0,Y 125.966,Z 671.037,A -85,B 0,C 180,E1 -30947.525,E2 -30947.525} C_VEL
LIN {X 0,Y 132.09,Z 656.392,A -85,B 0,C 180,E1 -30947.634,E2 -30947.634} C_VEL
LIN {X 0,Y 136.984,Z 640.856,A -85,B 0,C 180,E1 -30947.742,E2 -30947.742} C_VEL
LIN {X 0,Y 139.307,Z 630.874,A -85,B 0,C 180,E1 -30947.796,E2 -30947.796} C_VEL
LIN {X 0,Y 139.329,Z 630.812,A -85,B 0,C 180,E1 -30949.947,E2 -30949.947} C_VEL
LIN {X 0,Y 135.59,Z 645.791,A -85,B 0,C 180,E1 -30950.011,E2 -30950.011} C_VEL
LIN {X 0,Y 130.52,Z 660.5,A -85,B 0,C 180,E1 -30949.975,E2 -30949.975} C_VEL
LIN {X 0,Y 124.002,Z 675.071,A -85,B 0,C 180,E1 -30949.988,E2 -30949.988} C_VEL
LIN {X 0,Y 116.424,Z 688.612,A -85,B 0,C 180,E1 -30949.906,E2 -30949.906} C_VEL
LIN {X 0,Y 108.874,Z 699.859,A -85,B 0,C 180,E1 -30949.88,E2 -30949.88} C_VEL
LIN {X 0,Y 99.946,Z 711.137,A -85,B 0,C 180,E1 -30949.891,E2 -30949.891} C_VEL
LIN {X 0,Y 89.227,Z 722.503,A -85,B 0,C 180,E1 -30949.931,E2 -30949.931} C_VEL
LIN {X 0,Y 76.753,Z 733.472,A -85,B 0,C 180,E1 -30949.86,E2 -30949.86} C_VEL
LIN {X 0,Y 64.22,Z 742.63,A -85,B 0,C 180,E1 -30950.057,E2 -30950.057} C_VEL
LIN {X 0,Y 51.735,Z 750.19,A -85,B 0,C 180,E1 -30950.046,E2 -30950.046} C_VEL
LIN {X 0,Y 40.195,Z 755.932,A -85,B 0,C 180,E1 -30949.928,E2 -30949.928} C_VEL
LIN {X 0,Y 25.008,Z 762.004,A -85,B 0,C 180,E1 -30949.654,E2 -30949.654} C_VEL
LIN {X 0,Y 21.463,Z 763.201,A -85,B 0,C 180,E1 -30949.264,E2 -30949.264} C_VEL
LIN {X 0,Y 21.664,Z 763.119,A -85,B 0,C 180,E1 -30946.758,E2 -30946.758} C_VEL
LIN {X 0,Y 36.203,Z 757.664,A -85,B 0,C 180,E1 -30946.102,E2 -30946.102} C_VEL
LIN {X 0,Y 50.648,Z 750.705,A -85,B 0,C 180,E1 -30946.264,E2 -30946.264} C_VEL
LIN {X 0,Y 56.04,Z 747.642,A -85,B 0,C 180,E1 -30946.39,E2 -30946.39} C_VEL
LIN {X 0,Y 56.04,Z 747.642,A -85,B 0,C 180,E1 -30946.39,E2 -30946.39}

QRS_NEXT_CUT()

QRS_NEXT()
QRS_HOME()

END
